KUKA KRL program: MyProgram_033().src

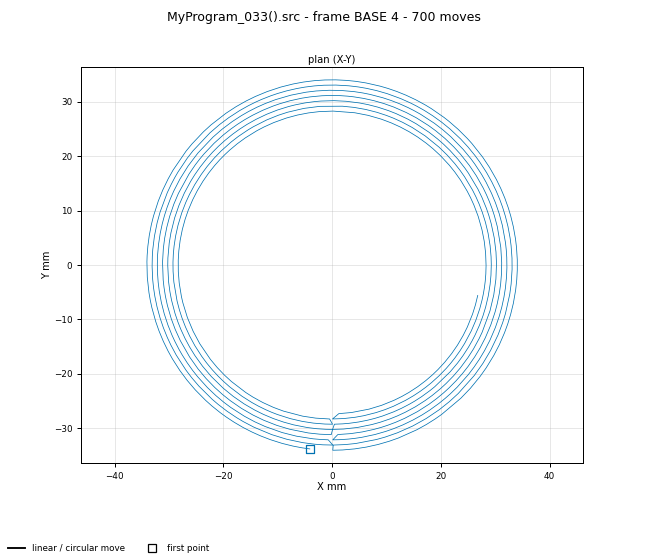
[picture p0: tool path of MyProgram_033().src in frame BASE 4, 700 of 700 moves have a stored position in this frame; points joined in program order, loops and branches not executed]
&ACCESS RVP
&REL 1
&PARAM TEMPLATE = C:\KRC\Roboter\Template\vorgabe
&PARAM EDITMASK = *
DEF MyProgram_033()
; ---- Setting reference (Base) ----
$BASE = BASE_DATA[4]

; --------------------------
; ---- Setting tool (TCP) ----
$TOOL = TOOL_DATA[3]
; --------------------------

$VEL.CP = VEL_APROX_PRINT
Startdeposition()
$VEL.CP = VEL_PRINT
LIN {X -4.1011,Y -33.8077,Z 60,A -103.7519,B 24.8568,C -2.7608,E1 24.9802,E2 -893.1526} C_DIS
LIN {X -5.5425,Y -33.6018,Z 60,A -106.5325,B 24.8572,C -2.7577,E1 24.9725,E2 -890.3623} C_DIS
LIN {X -7.2068,Y -33.2842,Z 60,A -109.5413,B 24.8572,C -2.7571,E1 24.9643,E2 -887.3486} C_DIS
LIN {X -9.1844,Y -32.7935,Z 60,A -113.0761,B 24.8572,C -2.7579,E1 24.9547,E2 -883.8105} C_DIS
LIN {X -11.3943,Y -32.093,Z 60,A -117.2451,B 24.8572,C -2.7582,E1 24.9437,E2 -879.6342} C_DIS
LIN {X -13.2172,Y -31.3861,Z 60,A -119.8941,B 24.8561,C -2.7679,E1 24.9369,E2 -877.0026} C_DIS
LIN {X -14.7733,Y -30.6845,Z 60,A -123.1754,B 24.8561,C -2.767,E1 24.9285,E2 -873.7109} C_DIS
LIN {X -16.3966,Y -29.8493,Z 60,A -126.0085,B 24.8555,C -2.7732,E1 24.9216,E2 -870.8848} C_DIS
LIN {X -18.0247,Y -28.8947,Z 60,A -129.5512,B 24.8555,C -2.7742,E1 24.9131,E2 -867.3333} C_DIS
LIN {X -19.4848,Y -27.931,Z 60,A -132.0562,B 24.8545,C -2.783,E1 24.9073,E2 -864.8412} C_DIS
LIN {X -20.5573,Y -27.1516,Z 60,A -134.7533,B 24.8545,C -2.7823,E1 24.9013,E2 -862.1327} C_DIS
LIN {X -22.102,Y -25.9094,Z 60,A -137.784,B 24.8536,C -2.7913,E1 24.8948,E2 -859.1119} C_DIS
LIN {X -23.2509,Y -24.8836,Z 60,A -140.7805,B 24.8536,C -2.7926,E1 24.8886,E2 -856.1064} C_DIS
LIN {X -25.1661,Y -22.9451,Z 60,A -144.9973,B 24.8521,C -2.8056,E1 24.8805,E2 -851.9024} C_DIS
LIN {X -26.6648,Y -21.1845,Z 60,A -149.0986,B 24.8514,C -2.8125,E1 24.8732,E2 -847.7987} C_DIS
LIN {X -28.0034,Y -19.3806,Z 60,A -153.0848,B 24.8506,C -2.8198,E1 24.8667,E2 -843.8106} C_DIS
LIN {X -29.3744,Y -17.2323,Z 60,A -156.9438,B 24.8491,C -2.8344,E1 24.861,E2 -839.9668} C_DIS
LIN {X -30.1456,Y -15.8438,Z 60,A -159.4556,B 24.8482,C -2.8429,E1 24.8577,E2 -837.4619} C_DIS
LIN {X -31.038,Y -14.0154,Z 60,A -163.101,B 24.8474,C -2.8503,E1 24.8533,E2 -833.8145} C_DIS
LIN {X -31.8171,Y -12.1432,Z 60,A -166.7902,B 24.8466,C -2.8576,E1 24.8495,E2 -830.1221} C_DIS
LIN {X -32.4094,Y -10.4598,Z 60,A -170.2484,B 24.846,C -2.8626,E1 24.8465,E2 -826.656} C_DIS
LIN {X -33.145,Y -7.823,Z 60,A -174.1454,B 24.8439,C -2.882,E1 24.8437,E2 -822.7829} C_DIS
LIN {X -33.441,Y -6.4408,Z 60,A -176.5305,B 24.8432,C -2.8891,E1 24.8424,E2 -820.4008} C_DIS
LIN {X -33.6768,Y -5.0685,Z 60,A -179.4437,B 24.8429,C -2.8917,E1 24.8411,E2 -817.4763} C_DIS
LIN {X -33.9818,Y -2.2443,Z 60,A 175.55,B 24.8415,C -2.9046,E1 24.8399,E2 -812.4709} C_DIS
LIN {X -34.0507,Y 0.5917,Z 60,A 171.6162,B 24.8391,C -2.9263,E1 24.8399,E2 -808.5652} C_DIS
LIN {X -34.0099,Y 1.7604,Z 60,A 169.3433,B 24.8387,C -2.93,E1 24.8401,E2 -806.2875} C_DIS
LIN {X -33.8822,Y 3.4352,Z 60,A 166.5069,B 24.8377,C -2.9387,E1 24.8408,E2 -803.455} C_DIS
LIN {X -33.6225,Y 5.4145,Z 60,A 163.0669,B 24.8366,C -2.9485,E1 24.8422,E2 -800.018} C_DIS
LIN {X -33.2455,Y 7.3857,Z 60,A 159.4228,B 24.8357,C -2.9568,E1 24.8443,E2 -796.3723} C_DIS
LIN {X -32.8452,Y 8.998,Z 60,A 156.7201,B 24.8347,C -2.9662,E1 24.8462,E2 -793.6762} C_DIS
LIN {X -31.9703,Y 11.7339,Z 60,A 151.2142,B 24.8336,C -2.9753,E1 24.8512,E2 -788.161} C_DIS
LIN {X -31.1372,Y 13.7944,Z 60,A 147.9434,B 24.832,C -2.9901,E1 24.8548,E2 -784.9074} C_DIS
LIN {X -30.1384,Y 15.8574,Z 60,A 144.453,B 24.8304,C -3.0042,E1 24.8591,E2 -781.4321} C_DIS
LIN {X -29.2375,Y 17.4636,Z 60,A 140.1056,B 24.8305,C -3.0026,E1 24.8654,E2 -777.0583} C_DIS
LIN {X -26.8529,Y 20.9464,Z 60,A 134.1639,B 24.8273,C -3.0311,E1 24.875,E2 -771.1559} C_DIS
LIN {X -25.7967,Y 22.2333,Z 60,A 130.7426,B 24.8271,C -3.0329,E1 24.8812,E2 -767.7231} C_DIS
LIN {X -23.6637,Y 24.4914,Z 60,A 125.988,B 24.8252,C -3.0493,E1 24.8904,E2 -762.9876} C_DIS
LIN {X -22.2685,Y 25.7663,Z 60,A 122.1842,B 24.825,C -3.0508,E1 24.8984,E2 -759.1724} C_DIS
LIN {X -19.5115,Y 27.912,Z 60,A 116.7582,B 24.8232,C -3.0668,E1 24.9105,E2 -753.7652} C_DIS
LIN {X -17.6615,Y 29.1182,Z 60,A 113.1214,B 24.8223,C -3.0743,E1 24.9191,E2 -750.1348} C_DIS
LIN {X -15.826,Y 30.1549,Z 60,A 109.4298,B 24.8218,C -3.0789,E1 24.9281,E2 -746.4435} C_DIS
LIN {X -14.122,Y 30.9898,Z 60,A 106.4786,B 24.821,C -3.086,E1 24.9356,E2 -743.5019} C_DIS
LIN {X -11.9367,Y 31.8948,Z 60,A 102.2584,B 24.8206,C -3.089,E1 24.9465,E2 -739.2795} C_DIS
LIN {X -9.4384,Y 32.7218,Z 60,A 97.5577,B 24.8204,C -3.0912,E1 24.9591,E2 -734.5758} C_DIS
LIN {X -7.1696,Y 33.2922,Z 60,A 94.1206,B 24.8193,C -3.0998,E1 24.9684,E2 -731.1548} C_DIS
LIN {X -5.2376,Y 33.6506,Z 60,A 90.6316,B 24.8193,C -3.1003,E1 24.978,E2 -727.6635} C_DIS
LIN {X -3.27,Y 33.8982,Z 60,A 87.248,B 24.8191,C -3.1015,E1 24.9874,E2 -724.2808} C_DIS
LIN {X -1.3206,Y 34.0299,Z 60,A 83.9345,B 24.8191,C -3.1024,E1 24.9966,E2 -720.9685} C_DIS
LIN {X 0.6663,Y 34.0493,Z 60,A 80.7843,B 24.8187,C -3.1051,E1 25.0054,E2 -717.825} C_DIS
LIN {X 2.7045,Y 33.9479,Z 60,A 77.3953,B 24.8187,C -3.1056,E1 25.0148,E2 -714.4386} C_DIS
LIN {X 4.3939,Y 33.771,Z 60,A 74.5416,B 24.8187,C -3.1052,E1 25.0227,E2 -711.5859} C_DIS
LIN {X 6.2336,Y 33.4806,Z 60,A 70.9287,B 24.8195,C -3.0986,E1 25.0327,E2 -707.9612} C_DIS
LIN {X 8.817,Y 32.8943,Z 60,A 66.9146,B 24.8192,C -3.1013,E1 25.0435,E2 -703.9594} C_DIS
LIN {X 10.2829,Y 32.4658,Z 60,A 64.544,B 24.8192,C -3.1018,E1 25.0499,E2 -701.5942} C_DIS
LIN {X 11.8741,Y 31.9182,Z 60,A 61.4166,B 24.8198,C -3.0958,E1 25.0581,E2 -698.4589} C_DIS
LIN {X 13.5855,Y 31.2283,Z 60,A 58.3959,B 24.8201,C -3.0937,E1 25.0659,E2 -695.4401} C_DIS
LIN {X 15.3952,Y 30.3775,Z 60,A 54.9755,B 24.8206,C -3.0889,E1 25.0745,E2 -692.0176} C_DIS
LIN {X 17.1475,Y 29.4242,Z 60,A 51.9399,B 24.8206,C -3.0884,E1 25.0819,E2 -688.9897} C_DIS
LIN {X 18.2192,Y 28.7727,Z 60,A 49.141,B 24.8221,C -3.0765,E1 25.0885,E2 -686.1715} C_DIS
LIN {X 20.5404,Y 27.1644,Z 60,A 45.1493,B 24.8218,C -3.0784,E1 25.0975,E2 -682.1983} C_DIS
LIN {X 21.455,Y 26.4477,Z 60,A 42.9139,B 24.8227,C -3.0713,E1 25.1024,E2 -679.9543} C_DIS
LIN {X 23.1922,Y 24.9385,Z 60,A 38.6625,B 24.8241,C -3.0588,E1 25.1113,E2 -675.6903} C_DIS
LIN {X 24.8778,Y 23.2567,Z 60,A 35.3372,B 24.8241,C -3.0594,E1 25.1177,E2 -672.3807} C_DIS
LIN {X 25.686,Y 22.3614,Z 60,A 32.55,B 24.8257,C -3.0448,E1 25.1229,E2 -669.5713} C_DIS
LIN {X 27.6713,Y 19.852,Z 60,A 28.2174,B 24.8255,C -3.0464,E1 25.1303,E2 -665.2631} C_DIS
LIN {X 28.9223,Y 17.9798,Z 60,A 23.4081,B 24.8282,C -3.0228,E1 25.1376,E2 -660.422} C_DIS
LIN {X 30.1935,Y 15.7523,Z 60,A 19.4635,B 24.829,C -3.0166,E1 25.1429,E2 -656.4831} C_DIS
LIN {X 31.019,Y 14.0575,Z 60,A 16.5637,B 24.8295,C -3.0117,E1 25.1463,E2 -653.5874} C_DIS
LIN {X 31.744,Y 12.3327,Z 60,A 13.1959,B 24.8309,C -2.9997,E1 25.1499,E2 -650.2098} C_DIS
LIN {X 32.3816,Y 10.5466,Z 60,A 10.2406,B 24.8315,C -2.9938,E1 25.1525,E2 -647.2573} C_DIS
LIN {X 32.847,Y 8.9926,Z 60,A 7.5063,B 24.8325,C -2.9857,E1 25.1546,E2 -644.5194} C_DIS
LIN {X 33.3186,Y 7.0474,Z 60,A 3.8113,B 24.8341,C -2.9709,E1 25.1569,E2 -640.8108} C_DIS
LIN {X 33.7159,Y 4.7991,Z 60,A 0.1976,B 24.8351,C -2.9624,E1 25.1585,E2 -637.1983} C_DIS
LIN {X 33.9025,Y 3.2253,Z 60,A -2.4984,B 24.836,C -2.9537,E1 25.1593,E2 -634.4977} C_DIS
LIN {X 34.0412,Y 0.9926,Z 60,A -6.0206,B 24.837,C -2.9455,E1 25.1598,E2 -630.977} C_DIS
LIN {X 34.043,Y -0.9308,Z 60,A -9.3922,B 24.8383,C -2.9334,E1 25.1596,E2 -627.5968} C_DIS
LIN {X 33.9493,Y -2.6804,Z 60,A -12.2431,B 24.8392,C -2.9256,E1 25.1591,E2 -624.7443} C_DIS
LIN {X 33.7459,Y -4.5841,Z 60,A -15.5123,B 24.8404,C -2.9148,E1 25.158,E2 -621.4688} C_DIS
LIN {X 33.3196,Y -7.0427,Z 60,A -19.7936,B 24.8419,C -2.9005,E1 25.1558,E2 -617.1788} C_DIS
LIN {X 32.8125,Y -9.1163,Z 60,A -23.0848,B 24.8427,C -2.8938,E1 25.1535,E2 -613.8906} C_DIS
LIN {X 32.296,Y -10.8043,Z 60,A -25.7379,B 24.8431,C -2.8893,E1 25.1512,E2 -611.2421} C_DIS
LIN {X 31.7073,Y -12.4251,Z 60,A -28.7099,B 24.8442,C -2.8796,E1 25.1483,E2 -608.2636} C_DIS
LIN {X 30.7314,Y -14.6755,Z 60,A -33.9408,B 24.8472,C -2.8517,E1 25.1422,E2 -602.9951} C_DIS
LIN {X 29.7216,Y -16.626,Z 60,A -37.262,B 24.8478,C -2.8465,E1 25.1378,E2 -599.6788} C_DIS
LIN {X 28.3176,Y -18.9173,Z 60,A -41.1609,B 24.8482,C -2.8428,E1 25.1319,E2 -595.7907} C_DIS
LIN {X 27.2015,Y -20.4909,Z 60,A -44.1382,B 24.8487,C -2.8379,E1 25.1271,E2 -592.8163} C_DIS
LIN {X 25.4199,Y -22.6633,Z 60,A -49.9904,B 24.8516,C -2.8103,E1 25.1164,E2 -586.9256} C_DIS
LIN {X 23.6533,Y -24.5014,Z 60,A -54.523,B 24.853,C -2.797,E1 25.1074,E2 -582.3803} C_DIS
LIN {X 20.127,Y -27.4718,Z 60,A -60.5922,B 24.8524,C -2.8031,E1 25.0943,E2 -576.3485} C_DIS
LIN {X 18.9319,Y -28.3082,Z 60,A -63.281,B 24.8532,C -2.7951,E1 25.0881,E2 -573.65} C_DIS
LIN {X 17.3293,Y -29.3171,Z 60,A -67.2414,B 24.8549,C -2.7791,E1 25.0786,E2 -569.664} C_DIS
LIN {X 15.5543,Y -30.2963,Z 60,A -70.9708,B 24.8559,C -2.7694,E1 25.0693,E2 -565.922} C_DIS
LIN {X 12.179,Y -31.8037,Z 60,A -76.2659,B 24.8556,C -2.7723,E1 25.0558,E2 -560.6462} C_DIS
LIN {X 10.5249,Y -32.3887,Z 60,A -79.589,B 24.8565,C -2.764,E1 25.0469,E2 -557.31} C_DIS
LIN {X 8.4575,Y -32.9886,Z 60,A -83.2845,B 24.857,C -2.7593,E1 25.037,E2 -553.6093} C_DIS
LIN {X 6.2909,Y -33.4695,Z 60,A -86.7215,B 24.857,C -2.7598,E1 25.0276,E2 -550.1776} C_DIS
LIN {X 4.1516,Y -33.8017,Z 60,A -90.2648,B 24.857,C -2.7585,E1 25.0178,E2 -546.6345} C_DIS
LIN {X 1.9064,Y -34.0016,Z 60,A -94.0756,B 24.8573,C -2.7566,E1 25.0072,E2 -542.8209} C_DIS
LIN {X 0.1202,Y -34.0515,Z 60,A -95.9136,B 24.8559,C -2.7694,E1 25.0021,E2 -541.0138} C_DIS
Enddeposition()
LIN {X 0.1202,Y -34.0515,Z 60,A -95.9136,B 24.8559,C -2.7694,E1 25.0021,E2 -541.0138} C_DIS
Startdeposition()
$VEL.CP = VEL_PRINT
LIN {X 0.2045,Y -33.097,Z 60,A -95.4369,B 24.8538,C -2.7896,E1 25.0036,E2 -541.5385} C_DIS
LIN {X 2.3595,Y -33.0129,Z 60,A -91.3479,B 24.8532,C -2.7953,E1 25.015,E2 -545.6395} C_DIS
LIN {X 4.3325,Y -32.8127,Z 60,A -87.4957,B 24.8525,C -2.8025,E1 25.0257,E2 -549.5057} C_DIS
LIN {X 8.1456,Y -32.0792,Z 60,A -81.9514,B 24.8534,C -2.7939,E1 25.0408,E2 -555.0225} C_DIS
LIN {X 9.7251,Y -31.6363,Z 60,A -78.376,B 24.8521,C -2.8062,E1 25.0504,E2 -558.6209} C_DIS
LIN {X 12.006,Y -30.843,Z 60,A -74.0706,B 24.8513,C -2.8132,E1 25.0617,E2 -562.9339} C_DIS
LIN {X 14.8198,Y -29.5942,Z 60,A -69.0859,B 24.8509,C -2.8169,E1 25.0743,E2 -567.9146} C_DIS
LIN {X 17.289,Y -28.2232,Z 60,A -63.6869,B 24.8493,C -2.8323,E1 25.0874,E2 -573.3336} C_DIS
LIN {X 19.6801,Y -26.6116,Z 60,A -59.6968,B 24.8497,C -2.8288,E1 25.0964,E2 -577.3018} C_DIS
LIN {X 21.5621,Y -25.1105,Z 60,A -54.3541,B 24.847,C -2.8538,E1 25.108,E2 -582.6832} C_DIS
LIN {X 23.1978,Y -23.6076,Z 60,A -50.3874,B 24.8458,C -2.8645,E1 25.1159,E2 -586.6586} C_DIS
LIN {X 26.126,Y -20.3201,Z 60,A -43.8899,B 24.8455,C -2.868,E1 25.1276,E2 -593.1349} C_DIS
LIN {X 27.705,Y -18.1078,Z 60,A -38.537,B 24.8431,C -2.8899,E1 25.1361,E2 -598.5131} C_DIS
LIN {X 29.1251,Y -15.7222,Z 60,A -33.8097,B 24.8417,C -2.9024,E1 25.1426,E2 -603.2454} C_DIS
LIN {X 30.4955,Y -12.8635,Z 60,A -28.9128,B 24.8409,C -2.91,E1 25.1482,E2 -608.1339} C_DIS
LIN {X 31.3542,Y -10.6002,Z 60,A -24.761,B 24.8395,C -2.9221,E1 25.1522,E2 -612.2911} C_DIS
LIN {X 31.8641,Y -8.9501,Z 60,A -21.1192,B 24.8375,C -2.9407,E1 25.155,E2 -615.9559} C_DIS
LIN {X 32.6625,Y -5.3501,Z 60,A -15.7724,B 24.837,C -2.9455,E1 25.1579,E2 -621.283} C_DIS
LIN {X 32.9129,Y -3.4907,Z 60,A -11.951,B 24.8349,C -2.964,E1 25.1592,E2 -625.1255} C_DIS
LIN {X 33.0886,Y -0.7895,Z 60,A -7.3415,B 24.8334,C -2.9775,E1 25.1598,E2 -629.7397} C_DIS
LIN {X 33.0726,Y 1.2789,Z 60,A -3.8158,B 24.8322,C -2.9879,E1 25.1595,E2 -633.269} C_DIS
LIN {X 32.9048,Y 3.567,Z 60,A -0.295,B 24.8316,C -2.9937,E1 25.1586,E2 -636.7827} C_DIS
LIN {X 32.7236,Y 4.9627,Z 60,A 2.3683,B 24.8303,C -3.0044,E1 25.1576,E2 -639.4557} C_DIS
LIN {X 32.3321,Y 7.0767,Z 60,A 5.9021,B 24.8294,C -3.013,E1 25.1557,E2 -642.9891} C_DIS
LIN {X 31.8536,Y 8.9878,Z 60,A 9.2415,B 24.8283,C -3.0221,E1 25.1533,E2 -646.3309} C_DIS
LIN {X 31.334,Y 10.6598,Z 60,A 12.4134,B 24.8271,C -3.0329,E1 25.1505,E2 -649.5104} C_DIS
LIN {X 30.8145,Y 12.0789,Z 60,A 14.7067,B 24.8268,C -3.0358,E1 25.1483,E2 -651.7979} C_DIS
LIN {X 30.1671,Y 13.6158,Z 60,A 17.9721,B 24.8252,C -3.0492,E1 25.1446,E2 -655.077} C_DIS
LIN {X 29.3671,Y 15.2653,Z 60,A 20.8782,B 24.8247,C -3.054,E1 25.141,E2 -657.9791} C_DIS
LIN {X 28.3881,Y 17.0175,Z 60,A 24.7982,B 24.8229,C -3.0692,E1 25.1355,E2 -661.9149} C_DIS
LIN {X 27.1221,Y 18.9699,Z 60,A 27.9977,B 24.8231,C -3.0679,E1 25.1305,E2 -665.0953} C_DIS
LIN {X 26.2731,Y 20.1291,Z 60,A 31.0095,B 24.8216,C -3.0809,E1 25.1255,E2 -668.1236} C_DIS
LIN {X 24.9894,Y 21.7024,Z 60,A 34.3231,B 24.8209,C -3.0861,E1 25.1195,E2 -671.4345} C_DIS
LIN {X 23.6198,Y 23.1855,Z 60,A 38.4346,B 24.8191,C -3.1018,E1 25.1115,E2 -675.5653} C_DIS
LIN {X 21.6787,Y 25.0098,Z 60,A 42.4056,B 24.8191,C -3.1023,E1 25.1034,E2 -679.5217} C_DIS
LIN {X 20.1341,Y 26.2693,Z 60,A 46.2217,B 24.8178,C -3.1132,E1 25.095,E2 -683.3494} C_DIS
LIN {X 18.4879,Y 27.4526,Z 60,A 49.4342,B 24.8176,C -3.1151,E1 25.0876,E2 -686.5553} C_DIS
LIN {X 16.9247,Y 28.4433,Z 60,A 52.4596,B 24.8173,C -3.1176,E1 25.0804,E2 -689.577} C_DIS
LIN {X 15.6004,Y 29.1906,Z 60,A 54.8557,B 24.8172,C -3.1181,E1 25.0746,E2 -691.9675} C_DIS
LIN {X 14.4137,Y 29.7944,Z 60,A 57.4788,B 24.8164,C -3.1249,E1 25.068,E2 -694.5996} C_DIS
LIN {X 12.61,Y 30.6015,Z 60,A 61.2733,B 24.8154,C -3.133,E1 25.0582,E2 -698.4043} C_DIS
LIN {X 10.1317,Y 31.5084,Z 60,A 65.3664,B 24.8157,C -3.1312,E1 25.0475,E2 -702.4849} C_DIS
LIN {X 8.2097,Y 32.063,Z 60,A 69.151,B 24.8149,C -3.1371,E1 25.0373,E2 -706.2776} C_DIS
LIN {X 6.3041,Y 32.4916,Z 60,A 72.3612,B 24.815,C -3.1367,E1 25.0285,E2 -709.4826} C_DIS
LIN {X 4.8128,Y 32.7461,Z 60,A 74.7387,B 24.8152,C -3.1347,E1 25.022,E2 -711.8532} C_DIS
LIN {X 3.0706,Y 32.9547,Z 60,A 78.3371,B 24.8144,C -3.1414,E1 25.0119,E2 -715.4651} C_DIS
LIN {X 0.6892,Y 33.0906,Z 60,A 82.3493,B 24.8146,C -3.1398,E1 25.0008,E2 -719.4724} C_DIS
LIN {X -1.5064,Y 33.0631,Z 60,A 85.9149,B 24.8151,C -3.1362,E1 24.9908,E2 -723.0299} C_DIS
LIN {X -3.2719,Y 32.9353,Z 60,A 89.2096,B 24.8149,C -3.1372,E1 24.9817,E2 -726.3286} C_DIS
LIN {X -5.02,Y 32.7148,Z 60,A 91.7867,B 24.8157,C -3.1304,E1 24.9746,E2 -728.8915} C_DIS
LIN {X -6.5185,Y 32.4493,Z 60,A 94.6895,B 24.8157,C -3.1311,E1 24.9666,E2 -731.7991} C_DIS
LIN {X -8.3984,Y 32.0142,Z 60,A 98.2278,B 24.8157,C -3.13,E1 24.957,E2 -735.3397} C_DIS
LIN {X -10.0341,Y 31.5395,Z 60,A 100.7953,B 24.8166,C -3.123,E1 24.9502,E2 -737.8948} C_DIS
LIN {X -11.274,Y 31.118,Z 60,A 103.5496,B 24.8164,C -3.125,E1 24.9429,E2 -740.6594} C_DIS
LIN {X -12.9995,Y 30.4377,Z 60,A 106.309,B 24.8174,C -3.1162,E1 24.9358,E2 -743.404} C_DIS
LIN {X -14.1215,Y 29.9343,Z 60,A 108.4303,B 24.8178,C -3.113,E1 24.9304,E2 -745.5229} C_DIS
LIN {X -15.3884,Y 29.3025,Z 60,A 110.9912,B 24.8181,C -3.1101,E1 24.9241,E2 -748.0839} C_DIS
LIN {X -17.0304,Y 28.3798,Z 60,A 114.8593,B 24.8181,C -3.1101,E1 24.9147,E2 -751.9636} C_DIS
LIN {X -19.006,Y 27.0964,Z 60,A 118.1285,B 24.8199,C -3.095,E1 24.9072,E2 -755.2074} C_DIS
LIN {X -20.7047,Y 25.8224,Z 60,A 122.9494,B 24.8196,C -3.0977,E1 24.8965,E2 -760.0525} C_DIS
LIN {X -22.4758,Y 24.2961,Z 60,A 127.3905,B 24.8202,C -3.0921,E1 24.8874,E2 -764.4982} C_DIS
LIN {X -25.5874,Y 20.9946,Z 60,A 134.3352,B 24.8234,C -3.0648,E1 24.8745,E2 -771.4087} C_DIS
LIN {X -26.6205,Y 19.6678,Z 60,A 137.6287,B 24.8239,C -3.0605,E1 24.869,E2 -774.7075} C_DIS
LIN {X -28.3514,Y 17.0781,Z 60,A 142.2081,B 24.8264,C -3.0389,E1 24.8621,E2 -779.2585} C_DIS
LIN {X -28.9377,Y 16.0644,Z 60,A 144.4768,B 24.8268,C -3.0352,E1 24.859,E2 -781.5302} C_DIS
LIN {X -29.5648,Y 14.8797,Z 60,A 146.7395,B 24.8276,C -3.0281,E1 24.8561,E2 -783.7879} C_DIS
LIN {X -30.3082,Y 13.2994,Z 60,A 150.7686,B 24.8277,C -3.0275,E1 24.8515,E2 -787.8377} C_DIS
LIN {X -31.6393,Y 9.7155,Z 60,A 156.2309,B 24.8311,C -2.9982,E1 24.8465,E2 -793.2608} C_DIS
LIN {X -32.1756,Y 7.7552,Z 60,A 160.4111,B 24.8317,C -2.9927,E1 24.8436,E2 -797.4522} C_DIS
LIN {X -32.6737,Y 5.2775,Z 60,A 165.1809,B 24.8328,C -2.9822,E1 24.8412,E2 -802.2253} C_DIS
LIN {X -32.973,Y 2.8674,Z 60,A 168.4595,B 24.8352,C -2.9617,E1 24.8403,E2 -805.4743} C_DIS
LIN {X -33.057,Y 1.6305,Z 60,A 170.8713,B 24.8357,C -2.9571,E1 24.8399,E2 -807.8897} C_DIS
LIN {X -33.096,Y -0.2924,Z 60,A 174.4282,B 24.8366,C -2.9485,E1 24.8399,E2 -811.4474} C_DIS
LIN {X -32.9885,Y -2.6819,Z 60,A 178.201,B 24.8384,C -2.9327,E1 24.8404,E2 -815.2051} C_DIS
LIN {X -32.8369,Y -4.146,Z 60,A -179.0925,B 24.8391,C -2.9261,E1 24.8413,E2 -817.9121} C_DIS
LIN {X -32.594,Y -5.7529,Z 60,A -176.0974,B 24.8399,C -2.919,E1 24.8427,E2 -820.908} C_DIS
LIN {X -32.1918,Y -7.6888,Z 60,A -172.6651,B 24.841,C -2.9088,E1 24.8447,E2 -824.3361} C_DIS
LIN {X -31.643,Y -9.7037,Z 60,A -169.103,B 24.8422,C -2.8978,E1 24.8475,E2 -827.8923} C_DIS
LIN {X -31.0365,Y -11.4963,Z 60,A -165.5855,B 24.843,C -2.8904,E1 24.8508,E2 -831.412} C_DIS
LIN {X -30.3151,Y -13.2835,Z 60,A -162.7793,B 24.8445,C -2.8766,E1 24.8538,E2 -834.2009} C_DIS
LIN {X -29.6522,Y -14.7033,Z 60,A -159.5325,B 24.8448,C -2.8737,E1 24.8577,E2 -837.4584} C_DIS
LIN {X -28.67,Y -16.5374,Z 60,A -155.4519,B 24.8454,C -2.8684,E1 24.8633,E2 -841.5477} C_DIS
LIN {X -26.8802,Y -19.3109,Z 60,A -150.7238,B 24.8479,C -2.8457,E1 24.8706,E2 -846.2449} C_DIS
LIN {X -25.8421,Y -20.6801,Z 60,A -146.7435,B 24.8477,C -2.8477,E1 24.8775,E2 -850.2488} C_DIS
LIN {X -24.4962,Y -22.2575,Z 60,A -143.0433,B 24.8484,C -2.8408,E1 24.8844,E2 -853.9493} C_DIS
LIN {X -22.0604,Y -24.6738,Z 60,A -138.1883,B 24.8507,C -2.8189,E1 24.8941,E2 -858.7721} C_DIS
LIN {X -20.9813,Y -25.598,Z 60,A -135.1647,B 24.8507,C -2.8197,E1 24.9006,E2 -861.809} C_DIS
LIN {X -19.3358,Y -26.8623,Z 60,A -131.5019,B 24.8512,C -2.8143,E1 24.9088,E2 -865.4721} C_DIS
LIN {X -17.5879,Y -28.0377,Z 60,A -128.1825,B 24.8521,C -2.8056,E1 24.9165,E2 -868.7814} C_DIS
LIN {X -16.3357,Y -28.7859,Z 60,A -125.413,B 24.8523,C -2.8045,E1 24.9232,E2 -871.5566} C_DIS
LIN {X -14.3684,Y -29.8161,Z 60,A -120.9727,B 24.8521,C -2.8059,E1 24.9343,E2 -876.0121} C_DIS
LIN {X -11.0977,Y -31.1814,Z 60,A -114.7027,B 24.8525,C -2.8017,E1 24.9507,E2 -882.2853} C_DIS
LIN {X -8.3337,Y -32.0312,Z 60,A -109.9263,B 24.8531,C -2.7961,E1 24.9635,E2 -887.0559} C_DIS
LIN {X -5.4058,Y -32.6532,Z 60,A -105.0089,B 24.8536,C -2.7913,E1 24.9769,E2 -891.9672} C_DIS
LIN {X -3.2219,Y -32.9404,Z 60,A -101.8852,B 24.8545,C -2.7831,E1 24.9856,E2 -895.0735} C_DIS
LIN {X -1.6841,Y -33.0544,Z 60,A -98.863,B 24.8541,C -2.7871,E1 24.994,E2 -898.1063} C_DIS
LIN {X 0.1302,Y -33.0962,Z 60,A -97.1686,B 24.8557,C -2.7713,E1 24.9987,E2 -899.7633} C_DIS
Enddeposition()
LIN {X 0.1302,Y -33.0962,Z 60,A -97.1686,B 24.8557,C -2.7713,E1 24.9987,E2 -899.7633} C_DIS
Startdeposition()
$VEL.CP = VEL_PRINT
LIN {X -0.7153,Y -32.1318,Z 60,A -98.6258,B 24.854,C -2.7884,E1 24.9947,E2 -898.3466} C_DIS
LIN {X -2.0689,Y -32.0727,Z 60,A -100.8693,B 24.8538,C -2.7901,E1 24.9884,E2 -896.1066} C_DIS
LIN {X -3.5101,Y -31.9474,Z 60,A -103.7174,B 24.854,C -2.7874,E1 24.9805,E2 -893.2506} C_DIS
LIN {X -6.5606,Y -31.463,Z 60,A -110.1953,B 24.8549,C -2.7794,E1 24.9626,E2 -886.7468} C_DIS
LIN {X -9.1763,Y -30.8007,Z 60,A -114.641,B 24.8542,C -2.7861,E1 24.9507,E2 -882.3099} C_DIS
LIN {X -12.3035,Y -29.6913,Z 60,A -119.3861,B 24.8524,C -2.8026,E1 24.9384,E2 -877.5946} C_DIS
LIN {X -14.2126,Y -28.8258,Z 60,A -123.9875,B 24.8529,C -2.7986,E1 24.9267,E2 -872.972} C_DIS
LIN {X -16.1045,Y -27.8137,Z 60,A -128.1219,B 24.8526,C -2.8009,E1 24.9166,E2 -868.8309} C_DIS
LIN {X -18.6436,Y -26.1794,Z 60,A -132.797,B 24.8511,C -2.8156,E1 24.9058,E2 -864.1755} C_DIS
LIN {X -19.882,Y -25.2519,Z 60,A -135.745,B 24.8507,C -2.8187,E1 24.8993,E2 -861.2242} C_DIS
LIN {X -21.3807,Y -23.9963,Z 60,A -139.2884,B 24.8501,C -2.8247,E1 24.8918,E2 -857.6813} C_DIS
LIN {X -22.9252,Y -22.5252,Z 60,A -143.5033,B 24.8497,C -2.829,E1 24.8834,E2 -853.4589} C_DIS
LIN {X -24.7375,Y -20.5185,Z 60,A -147.746,B 24.848,C -2.8444,E1 24.8757,E2 -849.234} C_DIS
LIN {X -25.6401,Y -19.379,Z 60,A -150.286,B 24.8473,C -2.8509,E1 24.8713,E2 -846.6974} C_DIS
LIN {X -26.6364,Y -17.9848,Z 60,A -153.6792,B 24.8468,C -2.8556,E1 24.8659,E2 -843.2987} C_DIS
LIN {X -27.5573,Y -16.5395,Z 60,A -156.5093,B 24.8458,C -2.8652,E1 24.8618,E2 -840.477} C_DIS
LIN {X -28.1696,Y -15.4743,Z 60,A -158.7932,B 24.8452,C -2.8702,E1 24.8587,E2 -838.1931} C_DIS
LIN {X -28.8992,Y -14.0622,Z 60,A -161.3805,B 24.8442,C -2.8797,E1 24.8554,E2 -835.6148} C_DIS
LIN {X -29.4323,Y -12.9111,Z 60,A -164.1998,B 24.844,C -2.8816,E1 24.8522,E2 -832.7845} C_DIS
LIN {X -30.1822,Y -11.0442,Z 60,A -167.4588,B 24.8426,C -2.8943,E1 24.8489,E2 -829.5376} C_DIS
LIN {X -30.8706,Y -8.9417,Z 60,A -172.0182,B 24.8418,C -2.9012,E1 24.8452,E2 -824.9684} C_DIS
LIN {X -31.4046,Y -6.8329,Z 60,A -175.525,B 24.8403,C -2.9156,E1 24.843,E2 -821.4755} C_DIS
LIN {X -31.7843,Y -4.7678,Z 60,A -178.7753,B 24.8386,C -2.9306,E1 24.8414,E2 -818.2419} C_DIS
LIN {X -31.9804,Y -3.1964,Z 60,A 178.3793,B 24.8377,C -2.9391,E1 24.8405,E2 -815.3999} C_DIS
LIN {X -32.1078,Y -1.4183,Z 60,A 174.6768,B 24.837,C -2.9451,E1 24.8398,E2 -811.6893} C_DIS
LIN {X -32.1379,Y 0.2156,Z 60,A 172.0129,B 24.8358,C -2.956,E1 24.8398,E2 -809.0356} C_DIS
LIN {X -32.0787,Y 1.9696,Z 60,A 168.7941,B 24.8348,C -2.9651,E1 24.8402,E2 -805.8193} C_DIS
LIN {X -31.9124,Y 3.8118,Z 60,A 165.224,B 24.8338,C -2.9734,E1 24.8412,E2 -802.2476} C_DIS
LIN {X -31.6091,Y 5.8156,Z 60,A 161.6312,B 24.8326,C -2.9848,E1 24.8429,E2 -798.6608} C_DIS
LIN {X -31.2255,Y 7.6094,Z 60,A 158.365,B 24.8314,C -2.9949,E1 24.8449,E2 -795.3996} C_DIS
LIN {X -30.8172,Y 9.1232,Z 60,A 155.8063,B 24.8302,C -3.0052,E1 24.8468,E2 -792.8507} C_DIS
LIN {X -30.3452,Y 10.5875,Z 60,A 152.8019,B 24.8295,C -3.0116,E1 24.8495,E2 -789.8443} C_DIS
LIN {X -29.7422,Y 12.1789,Z 60,A 149.6558,B 24.8286,C -3.0198,E1 24.8527,E2 -786.7002} C_DIS
LIN {X -29.1245,Y 13.5905,Z 60,A 146.9426,B 24.8277,C -3.028,E1 24.8559,E2 -783.992} C_DIS
LIN {X -27.9696,Y 15.8309,Z 60,A 142.1992,B 24.8264,C -3.0389,E1 24.8621,E2 -779.2496} C_DIS
LIN {X -26.466,Y 18.2338,Z 60,A 136.5813,B 24.8253,C -3.0483,E1 24.8708,E2 -773.626} C_DIS
LIN {X -24.6789,Y 20.5889,Z 60,A 131.1092,B 24.824,C -3.0602,E1 24.8804,E2 -768.1569} C_DIS
LIN {X -21.891,Y 23.5318,Z 60,A 124.8467,B 24.8211,C -3.085,E1 24.8926,E2 -761.9269} C_DIS
LIN {X -20.2021,Y 24.9965,Z 60,A 120.4479,B 24.8205,C -3.0902,E1 24.902,E2 -757.5236} C_DIS
LIN {X -18.3745,Y 26.3691,Z 60,A 116.6627,B 24.8192,C -3.1007,E1 24.9106,E2 -753.7504} C_DIS
LIN {X -16.6745,Y 27.4755,Z 60,A 113.2127,B 24.8183,C -3.1088,E1 24.9187,E2 -750.3086} C_DIS
LIN {X -15.3521,Y 28.2359,Z 60,A 110.265,B 24.818,C -3.1113,E1 24.9259,E2 -747.3585} C_DIS
LIN {X -13.8092,Y 29.0216,Z 60,A 107.2908,B 24.8173,C -3.1171,E1 24.9333,E2 -744.3903} C_DIS
LIN {X -12.2881,Y 29.6966,Z 60,A 103.8696,B 24.8173,C -3.1171,E1 24.9421,E2 -740.9614} C_DIS
LIN {X -10.3903,Y 30.4138,Z 60,A 100.0066,B 24.8171,C -3.1193,E1 24.9523,E2 -737.0959} C_DIS
LIN {X -7.5813,Y 31.2322,Z 60,A 95.0969,B 24.8161,C -3.1274,E1 24.9655,E2 -732.1981} C_DIS
LIN {X -4.8177,Y 31.7765,Z 60,A 90.8046,B 24.8148,C -3.1382,E1 24.9772,E2 -727.9272} C_DIS
LIN {X -2.9177,Y 32.0061,Z 60,A 86.7045,B 24.8154,C -3.1332,E1 24.9887,E2 -723.8125} C_DIS
LIN {X -0.5298,Y 32.1352,Z 60,A 82.2698,B 24.8154,C -3.1327,E1 25.001,E2 -719.3761} C_DIS
LIN {X 1.6757,Y 32.0955,Z 60,A 78.4348,B 24.8154,C -3.134,E1 25.0117,E2 -715.5452} C_DIS
LIN {X 4.085,Y 31.8788,Z 60,A 74.6069,B 24.8148,C -3.1386,E1 25.0223,E2 -711.7307} C_DIS
LIN {X 5.6076,Y 31.6467,Z 60,A 71.8608,B 24.8148,C -3.1377,E1 25.0299,E2 -708.9853} C_DIS
LIN {X 6.9631,Y 31.3764,Z 60,A 68.9821,B 24.8156,C -3.132,E1 25.0378,E2 -706.0968} C_DIS
LIN {X 9.3593,Y 30.7464,Z 60,A 65.1991,B 24.8151,C -3.1363,E1 25.0479,E2 -702.33} C_DIS
LIN {X 10.8355,Y 30.2577,Z 60,A 62.148,B 24.8157,C -3.1308,E1 25.056,E2 -699.2719} C_DIS
LIN {X 12.413,Y 29.6454,Z 60,A 59.3663,B 24.8157,C -3.1306,E1 25.0632,E2 -696.4959} C_DIS
LIN {X 13.9702,Y 28.9444,Z 60,A 56.3307,B 24.8161,C -3.1272,E1 25.0709,E2 -693.46} C_DIS
LIN {X 15.0022,Y 28.4231,Z 60,A 54.1232,B 24.8166,C -3.1229,E1 25.0764,E2 -691.2484} C_DIS
LIN {X 16.2191,Y 27.7471,Z 60,A 51.0142,B 24.8179,C -3.112,E1 25.0839,E2 -688.1228} C_DIS
LIN {X 18.7648,Y 26.0924,Z 60,A 46.4958,B 24.8176,C -3.1143,E1 25.0944,E2 -683.6251} C_DIS
LIN {X 20.337,Y 24.8871,Z 60,A 42.3714,B 24.8192,C -3.1007,E1 25.1034,E2 -679.4837} C_DIS
LIN {X 21.8429,Y 23.5767,Z 60,A 38.334,B 24.8207,C -3.0878,E1 25.1118,E2 -675.432} C_DIS
LIN {X 24.0952,Y 21.2691,Z 60,A 33.1077,B 24.8214,C -3.0821,E1 25.1218,E2 -670.215} C_DIS
LIN {X 25.4626,Y 19.6114,Z 60,A 29.3914,B 24.8223,C -3.0747,E1 25.1282,E2 -666.4985} C_DIS
LIN {X 26.2596,Y 18.5308,Z 60,A 26.7666,B 24.8233,C -3.0659,E1 25.1325,E2 -663.8656} C_DIS
LIN {X 27.4745,Y 16.6753,Z 60,A 23.3272,B 24.8237,C -3.0626,E1 25.1376,E2 -660.4358} C_DIS
LIN {X 28.2947,Y 15.2435,Z 60,A 20.1887,B 24.8249,C -3.0523,E1 25.1419,E2 -657.2891} C_DIS
LIN {X 29.3,Y 13.2079,Z 60,A 15.7928,B 24.8267,C -3.0366,E1 25.1471,E2 -652.8797} C_DIS
LIN {X 30.0387,Y 11.4288,Z 60,A 12.6901,B 24.8273,C -3.0313,E1 25.1503,E2 -649.7817} C_DIS
LIN {X 30.7079,Y 9.4845,Z 60,A 8.9747,B 24.8286,C -3.0199,E1 25.1535,E2 -646.0605} C_DIS
LIN {X 31.3054,Y 7.2744,Z 60,A 4.5208,B 24.8305,C -3.0027,E1 25.1565,E2 -641.5916} C_DIS
LIN {X 31.8734,Y 4.1239,Z 60,A -0.0277,B 24.8307,C -3.0012,E1 25.1586,E2 -637.0661} C_DIS
LIN {X 32.0205,Y 2.7619,Z 60,A -2.7122,B 24.8319,C -2.9903,E1 25.1593,E2 -634.3717} C_DIS
LIN {X 32.1089,Y 1.3993,Z 60,A -5.2676,B 24.833,C -2.981,E1 25.1597,E2 -631.8096} C_DIS
LIN {X 32.1356,Y -0.5008,Z 60,A -8.7386,B 24.8343,C -2.9693,E1 25.1597,E2 -628.3314} C_DIS
LIN {X 32.0631,Y -2.2144,Z 60,A -11.8385,B 24.8354,C -2.9591,E1 25.1592,E2 -625.2259} C_DIS
LIN {X 31.8561,Y -4.2576,Z 60,A -15.3207,B 24.8364,C -2.9501,E1 25.1581,E2 -621.7431} C_DIS
LIN {X 31.589,Y -5.9233,Z 60,A -18.2147,B 24.8373,C -2.9423,E1 25.1567,E2 -618.8475} C_DIS
LIN {X 31.1975,Y -7.7244,Z 60,A -21.8323,B 24.8389,C -2.9276,E1 25.1544,E2 -615.216} C_DIS
LIN {X 30.7173,Y -9.4538,Z 60,A -24.5603,B 24.8393,C -2.9243,E1 25.1523,E2 -612.4958} C_DIS
LIN {X 30.0155,Y -11.4878,Z 60,A -28.9749,B 24.8414,C -2.9048,E1 25.1481,E2 -608.0598} C_DIS
LIN {X 29.0156,Y -13.8218,Z 60,A -33.5136,B 24.8429,C -2.8913,E1 25.1429,E2 -603.5139} C_DIS
LIN {X 28.0256,Y -15.7328,Z 60,A -36.8985,B 24.8435,C -2.8865,E1 25.1384,E2 -600.1352} C_DIS
LIN {X 27.0478,Y -17.36,Z 60,A -40.4846,B 24.8448,C -2.8744,E1 25.1331,E2 -596.5386} C_DIS
LIN {X 26.086,Y -18.7744,Z 60,A -43.1659,B 24.8451,C -2.8711,E1 25.1288,E2 -593.8626} C_DIS
LIN {X 25.0449,Y -20.1424,Z 60,A -46.9866,B 24.8471,C -2.8531,E1 25.1222,E2 -590.0173} C_DIS
LIN {X 23.0017,Y -22.4469,Z 60,A -51.78,B 24.8475,C -2.8488,E1 25.1131,E2 -585.2348} C_DIS
LIN {X 21.7425,Y -23.6688,Z 60,A -54.7202,B 24.848,C -2.844,E1 25.1072,E2 -582.2953} C_DIS
LIN {X 20.7778,Y -24.5195,Z 60,A -57.4236,B 24.8492,C -2.8337,E1 25.1014,E2 -579.5779} C_DIS
LIN {X 19.6299,Y -25.4483,Z 60,A -60.2652,B 24.85,C -2.8255,E1 25.0952,E2 -576.7274} C_DIS
LIN {X 17.9325,Y -26.6717,Z 60,A -63.4121,B 24.85,C -2.8255,E1 25.088,E2 -573.5913} C_DIS
LIN {X 16.5112,Y -27.5746,Z 60,A -66.6616,B 24.8509,C -2.8168,E1 25.0802,E2 -570.3317} C_DIS
LIN {X 14.8715,Y -28.4917,Z 60,A -69.9014,B 24.8514,C -2.8126,E1 25.0723,E2 -567.091} C_DIS
LIN {X 12.9889,Y -29.3982,Z 60,A -73.951,B 24.8524,C -2.803,E1 25.062,E2 -563.0289} C_DIS
LIN {X 11.2648,Y -30.1002,Z 60,A -76.7358,B 24.8522,C -2.8049,E1 25.0547,E2 -560.2549} C_DIS
LIN {X 9.8557,Y -30.5907,Z 60,A -79.6235,B 24.8528,C -2.799,E1 25.0471,E2 -557.3586} C_DIS
LIN {X 7.8541,Y -31.1647,Z 60,A -83.5946,B 24.8536,C -2.7921,E1 25.0363,E2 -553.3775} C_DIS
LIN {X 5.4947,Y -31.6662,Z 60,A -87.3055,B 24.8532,C -2.7953,E1 25.0262,E2 -549.6788} C_DIS
LIN {X 4.2567,Y -31.8562,Z 60,A -89.5663,B 24.8534,C -2.7935,E1 25.02,E2 -547.4156} C_DIS
LIN {X 2.9503,Y -32.0036,Z 60,A -92.0438,B 24.8537,C -2.7907,E1 25.0131,E2 -544.9331} C_DIS
LIN {X 1.3475,Y -32.111,Z 60,A -94.7433,B 24.8537,C -2.7914,E1 25.0055,E2 -542.2363} C_DIS
LIN {X 0.1197,Y -32.1384,Z 60,A -96.0087,B 24.8526,C -2.801,E1 25.0021,E2 -540.9938} C_DIS
Enddeposition()
LIN {X 0.1197,Y -32.1384,Z 60,A -96.0087,B 24.8526,C -2.801,E1 25.0021,E2 -540.9938} C_DIS
Startdeposition()
$VEL.CP = VEL_PRINT
LIN {X 1.0543,Y -31.1635,Z 60,A -93.7754,B 24.8502,C -2.8236,E1 25.0085,E2 -543.2805} C_DIS
LIN {X 3.3744,Y -30.998,Z 60,A -89.5002,B 24.85,C -2.8258,E1 25.0204,E2 -547.5584} C_DIS
LIN {X 5.5359,Y -30.6861,Z 60,A -85.3314,B 24.8495,C -2.8305,E1 25.0319,E2 -551.7342} C_DIS
LIN {X 7.684,Y -30.2194,Z 60,A -81.8831,B 24.8498,C -2.8274,E1 25.0412,E2 -555.1704} C_DIS
LIN {X 9.0101,Y -29.8513,Z 60,A -79.2571,B 24.8494,C -2.8313,E1 25.0483,E2 -557.8011} C_DIS
LIN {X 10.1777,Y -29.4734,Z 60,A -76.8788,B 24.849,C -2.8355,E1 25.0546,E2 -560.1848} C_DIS
LIN {X 11.6597,Y -28.9189,Z 60,A -73.9356,B 24.8485,C -2.8399,E1 25.0622,E2 -563.1318} C_DIS
LIN {X 13.3425,Y -28.1824,Z 60,A -70.3675,B 24.8477,C -2.8473,E1 25.0713,E2 -566.7085} C_DIS
LIN {X 15.6981,Y -26.9423,Z 60,A -65.1853,B 24.8464,C -2.8592,E1 25.084,E2 -571.904} C_DIS
LIN {X 17.8333,Y -25.5784,Z 60,A -61.1698,B 24.8464,C -2.8601,E1 25.0933,E2 -575.9082} C_DIS
LIN {X 19.2312,Y -24.545,Z 60,A -57.7676,B 24.8453,C -2.8694,E1 25.1009,E2 -579.32} C_DIS
LIN {X 20.5297,Y -23.4694,Z 60,A -55.0024,B 24.845,C -2.8719,E1 25.1067,E2 -582.0805} C_DIS
LIN {X 21.487,Y -22.5955,Z 60,A -52.4237,B 24.8442,C -2.88,E1 25.112,E2 -584.6677} C_DIS
LIN {X 22.8025,Y -21.2677,Z 60,A -49.0726,B 24.8434,C -2.8872,E1 25.1185,E2 -588.0213} C_DIS
LIN {X 23.9533,Y -19.9629,Z 60,A -45.8917,B 24.8425,C -2.895,E1 25.1243,E2 -591.2063} C_DIS
LIN {X 24.9987,Y -18.6374,Z 60,A -42.6484,B 24.8414,C -2.905,E1 25.1298,E2 -594.4579} C_DIS
LIN {X 26.2232,Y -16.8704,Z 60,A -39.0438,B 24.8408,C -2.9111,E1 25.1354,E2 -598.0592} C_DIS
LIN {X 27.2025,Y -15.2415,Z 60,A -35.1964,B 24.8392,C -2.9257,E1 25.1408,E2 -601.9213} C_DIS
LIN {X 28.1604,Y -13.3892,Z 60,A -31.4957,B 24.8381,C -2.935,E1 25.1454,E2 -605.6244} C_DIS
LIN {X 29.1727,Y -11.0089,Z 60,A -25.8485,B 24.8352,C -2.9615,E1 25.1513,E2 -611.3029} C_DIS
LIN {X 29.9671,Y -8.6178,Z 60,A -22.2384,B 24.8352,C -2.9615,E1 25.1542,E2 -614.8926} C_DIS
LIN {X 30.3516,Y -7.1441,Z 60,A -19.377,B 24.8341,C -2.9711,E1 25.1561,E2 -617.76} C_DIS
LIN {X 30.7297,Y -5.2897,Z 60,A -15.9973,B 24.833,C -2.9805,E1 25.1579,E2 -621.1423} C_DIS
LIN {X 30.987,Y -3.4768,Z 60,A -12.4884,B 24.8316,C -2.9931,E1 25.1591,E2 -624.6602} C_DIS
LIN {X 31.1456,Y -1.4774,Z 60,A -8.9261,B 24.8305,C -3.0029,E1 25.1597,E2 -628.2247} C_DIS
LIN {X 31.1787,Y 0.4322,Z 60,A -5.1764,B 24.8289,C -3.0172,E1 25.1597,E2 -631.9857} C_DIS
LIN {X 31.0092,Y 3.2713,Z 60,A 0.6137,B 24.8262,C -3.0411,E1 25.1583,E2 -637.7983} C_DIS
LIN {X 30.3685,Y 7.0725,Z 60,A 6.7788,B 24.8251,C -3.0499,E1 25.155,E2 -643.9483} C_DIS
LIN {X 29.8388,Y 9.0509,Z 60,A 10.1148,B 24.8245,C -3.0553,E1 25.1525,E2 -647.2777} C_DIS
LIN {X 29.4252,Y 10.316,Z 60,A 12.8631,B 24.8232,C -3.0664,E1 25.15,E2 -650.037} C_DIS
LIN {X 28.9382,Y 11.6118,Z 60,A 15.266,B 24.8226,C -3.0717,E1 25.1476,E2 -652.4391} C_DIS
LIN {X 28.385,Y 12.9065,Z 60,A 17.7697,B 24.8219,C -3.0778,E1 25.1448,E2 -654.9435} C_DIS
LIN {X 27.7748,Y 14.1718,Z 60,A 20.7476,B 24.8205,C -3.09,E1 25.141,E2 -657.9345} C_DIS
LIN {X 26.5119,Y 16.4138,Z 60,A 25.7099,B 24.8187,C -3.1053,E1 25.134,E2 -662.9077} C_DIS
LIN {X 25.2414,Y 18.3073,Z 60,A 29.6533,B 24.8179,C -3.1123,E1 25.1276,E2 -666.8483} C_DIS
LIN {X 23.6004,Y 20.379,Z 60,A 33.8746,B 24.8175,C -3.1153,E1 25.1202,E2 -671.0572} C_DIS
LIN {X 22.3378,Y 21.7556,Z 60,A 38.303,B 24.8152,C -3.1352,E1 25.1116,E2 -675.5137} C_DIS
LIN {X 20.7346,Y 23.2887,Z 60,A 41.897,B 24.8149,C -3.1372,E1 25.1043,E2 -679.0977} C_DIS
LIN {X 19.0515,Y 24.6845,Z 60,A 45.5264,B 24.8147,C -3.1396,E1 25.0964,E2 -682.7192} C_DIS
LIN {X 17.7132,Y 25.6612,Z 60,A 49.0782,B 24.8133,C -3.1508,E1 25.0883,E2 -686.2853} C_DIS
LIN {X 15.5118,Y 27.0493,Z 60,A 53.4233,B 24.8131,C -3.1525,E1 25.0779,E2 -690.6208} C_DIS
LIN {X 13.6406,Y 28.039,Z 60,A 57.9888,B 24.8116,C -3.1652,E1 25.0665,E2 -695.2041} C_DIS
LIN {X 11.3068,Y 29.0588,Z 60,A 62.0159,B 24.8119,C -3.1624,E1 25.0561,E2 -699.2153} C_DIS
LIN {X 9.4932,Y 29.7007,Z 60,A 65.6301,B 24.8115,C -3.1662,E1 25.0466,E2 -702.8314} C_DIS
LIN {X 7.6891,Y 30.2181,Z 60,A 68.9931,B 24.8113,C -3.1674,E1 25.0375,E2 -706.192} C_DIS
LIN {X 5.8076,Y 30.6355,Z 60,A 72.6037,B 24.8111,C -3.1697,E1 25.0276,E2 -709.8035} C_DIS
LIN {X 3.9305,Y 30.9327,Z 60,A 75.7558,B 24.8114,C -3.167,E1 25.019,E2 -712.9463} C_DIS
LIN {X 2.8125,Y 31.0543,Z 60,A 77.9312,B 24.8112,C -3.1684,E1 25.0129,E2 -715.1237} C_DIS
LIN {X 1.5034,Y 31.1447,Z 60,A 80.4289,B 24.8112,C -3.1692,E1 25.0059,E2 -717.6224} C_DIS
LIN {X -0.1002,Y 31.1809,Z 60,A 83.4801,B 24.8111,C -3.1698,E1 24.9974,E2 -720.6748} C_DIS
LIN {X -1.8789,Y 31.1243,Z 60,A 86.8709,B 24.8111,C -3.1699,E1 24.988,E2 -724.0666} C_DIS
LIN {X -4.0272,Y 30.9201,Z 60,A 90.6106,B 24.8116,C -3.1656,E1 24.9776,E2 -727.7982} C_DIS
LIN {X -5.5559,Y 30.682,Z 60,A 93.8473,B 24.8113,C -3.1674,E1 24.9687,E2 -731.0424} C_DIS
LIN {X -7.7892,Y 30.1922,Z 60,A 97.8112,B 24.8121,C -3.1613,E1 24.9579,E2 -734.9971} C_DIS
LIN {X -9.6775,Y 29.6415,Z 60,A 101.1922,B 24.8128,C -3.1552,E1 24.9489,E2 -738.3693} C_DIS
LIN {X -10.8512,Y 29.2319,Z 60,A 103.7873,B 24.8128,C -3.1552,E1 24.9421,E2 -740.9696} C_DIS
LIN {X -12.7741,Y 28.4444,Z 60,A 107.6457,B 24.8134,C -3.1501,E1 24.9322,E2 -744.825} C_DIS
LIN {X -14.6236,Y 27.5397,Z 60,A 111.1018,B 24.8145,C -3.1413,E1 24.9236,E2 -748.2692} C_DIS
LIN {X -16.0654,Y 26.7246,Z 60,A 114.4539,B 24.8148,C -3.1386,E1 24.9155,E2 -751.625} C_DIS
LIN {X -17.4051,Y 25.8715,Z 60,A 117.5237,B 24.8153,C -3.1345,E1 24.9084,E2 -754.6949} C_DIS
LIN {X -18.6835,Y 24.9641,Z 60,A 120.6562,B 24.8157,C -3.1308,E1 24.9013,E2 -757.8298} C_DIS
LIN {X -20.0124,Y 23.9121,Z 60,A 123.5953,B 24.8167,C -3.1227,E1 24.895,E2 -760.7607} C_DIS
LIN {X -21.6986,Y 22.3929,Z 60,A 127.9599,B 24.8176,C -3.1148,E1 24.8862,E2 -765.1243} C_DIS
LIN {X -23.5756,Y 20.4075,Z 60,A 132.2817,B 24.8197,C -3.097,E1 24.878,E2 -769.4226} C_DIS
LIN {X -24.3244,Y 19.5097,Z 60,A 134.6193,B 24.8201,C -3.093,E1 24.8739,E2 -771.7615} C_DIS
LIN {X -25.1742,Y 18.3991,Z 60,A 137.4932,B 24.8207,C -3.0886,E1 24.8691,E2 -774.6389} C_DIS
LIN {X -26.3057,Y 16.7417,Z 60,A 141.9609,B 24.8211,C -3.0847,E1 24.8623,E2 -779.1195} C_DIS
LIN {X -28.2686,Y 13.1585,Z 60,A 148.3078,B 24.8246,C -3.0543,E1 24.8542,E2 -785.4277} C_DIS
LIN {X -29.1071,Y 11.1808,Z 60,A 152.959,B 24.8254,C -3.0479,E1 24.8493,E2 -790.0893} C_DIS
LIN {X -29.8699,Y 8.9463,Z 60,A 157.2034,B 24.827,C -3.034,E1 24.8457,E2 -794.3248} C_DIS
LIN {X -30.3998,Y 6.9375,Z 60,A 160.9072,B 24.8284,C -3.0214,E1 24.8432,E2 -798.0202} C_DIS
LIN {X -30.7875,Y 4.9421,Z 60,A 164.6357,B 24.8297,C -3.0098,E1 24.8414,E2 -801.7429} C_DIS
LIN {X -31.0289,Y 3.0736,Z 60,A 168.4516,B 24.8307,C -3.0016,E1 24.8403,E2 -805.562} C_DIS
LIN {X -31.1766,Y 0.523,Z 60,A 173.4313,B 24.8321,C -2.989,E1 24.8398,E2 -810.5415} C_DIS
LIN {X -31.0598,Y -2.7524,Z 60,A 178.9441,B 24.8346,C -2.9665,E1 24.8407,E2 -816.0337} C_DIS
LIN {X -30.9108,Y -4.098,Z 60,A -178.6961,B 24.8356,C -2.958,E1 24.8415,E2 -818.387} C_DIS
LIN {X -30.6595,Y -5.6797,Z 60,A -175.9197,B 24.8367,C -2.9478,E1 24.8428,E2 -821.1556} C_DIS
LIN {X -30.2855,Y -7.4204,Z 60,A -172.4933,B 24.8377,C -2.9391,E1 24.8449,E2 -824.5814} C_DIS
LIN {X -29.5749,Y -9.878,Z 60,A -167.3676,B 24.8388,C -2.9286,E1 24.8491,E2 -829.7115} C_DIS
LIN {X -28.8495,Y -11.8311,Z 60,A -163.7196,B 24.8402,C -2.9164,E1 24.8528,E2 -833.3506} C_DIS
LIN {X -27.9126,Y -13.8982,Z 60,A -159.0014,B 24.841,C -2.9093,E1 24.8585,E2 -838.0775} C_DIS
LIN {X -26.1899,Y -16.9215,Z 60,A -152.6486,B 24.8428,C -2.8926,E1 24.8676,E2 -844.423} C_DIS
LIN {X -24.6366,Y -19.1131,Z 60,A -147.6997,B 24.8441,C -2.881,E1 24.8759,E2 -849.3679} C_DIS
LIN {X -23.1564,Y -20.8824,Z 60,A -143.8166,B 24.8454,C -2.8686,E1 24.883,E2 -853.239} C_DIS
LIN {X -21.5793,Y -22.5082,Z 60,A -139.481,B 24.8461,C -2.8616,E1 24.8916,E2 -857.5761} C_DIS
LIN {X -20.1344,Y -23.8097,Z 60,A -136.2421,B 24.8472,C -2.852,E1 24.8984,E2 -860.8047} C_DIS
LIN {X -18.7167,Y -24.9392,Z 60,A -132.7698,B 24.8477,C -2.8474,E1 24.906,E2 -864.2789} C_DIS
LIN {X -16.6708,Y -26.3504,Z 60,A -127.4414,B 24.8477,C -2.8474,E1 24.9185,E2 -869.6246} C_DIS
LIN {X -14.5491,Y -27.5788,Z 60,A -123.4787,B 24.8489,C -2.8364,E1 24.9282,E2 -873.5724} C_DIS
LIN {X -12.5599,Y -28.5402,Z 60,A -119.4427,B 24.8494,C -2.8317,E1 24.9384,E2 -877.6073} C_DIS
LIN {X -10.1755,Y -29.4741,Z 60,A -114.3827,B 24.8494,C -2.8311,E1 24.9517,E2 -882.6761} C_DIS
LIN {X -7.8468,Y -30.178,Z 60,A -109.6664,B 24.8494,C -2.8309,E1 24.9644,E2 -887.3991} C_DIS
LIN {X -4.3589,Y -30.8752,Z 60,A -103.6998,B 24.8503,C -2.8229,E1 24.9808,E2 -893.3527} C_DIS
LIN {X -2.231,Y -31.1011,Z 60,A -99.9597,B 24.8505,C -2.8207,E1 24.9912,E2 -897.0893} C_DIS
LIN {X -0.1621,Y -31.181,Z 60,A -95.8698,B 24.8501,C -2.8244,E1 25.0026,E2 -901.1883} C_DIS
LIN {X -0.1621,Y -31.181,Z 60,A -95.8698,B 24.8501,C -2.8244,E1 25.0026,E2 -901.1883} C_DIS
Enddeposition()
LIN {X 0.0842,Y -30.2228,Z 60,A -95.4358,B 24.8484,C -2.8405,E1 25.0039,E2 -901.6607} C_DIS
Startdeposition()
$VEL.CP = VEL_PRINT
LIN {X -1.136,Y -30.2018,Z 60,A -99.4718,B 24.8504,C -2.8222,E1 24.9925,E2 -897.5811} C_DIS
LIN {X -2.8098,Y -30.0921,Z 60,A -102.9498,B 24.8507,C -2.8193,E1 24.9828,E2 -894.0947} C_DIS
LIN {X -4.5561,Y -29.878,Z 60,A -106.5578,B 24.8509,C -2.8174,E1 24.9728,E2 -890.4791} C_DIS
LIN {X -7.0476,Y -29.3896,Z 60,A -111.0812,B 24.8504,C -2.8222,E1 24.9605,E2 -885.9617} C_DIS
LIN {X -8.9602,Y -28.8643,Z 60,A -114.8683,B 24.8501,C -2.8244,E1 24.9504,E2 -882.1737} C_DIS
LIN {X -10.8145,Y -28.2224,Z 60,A -118.4393,B 24.8497,C -2.829,E1 24.941,E2 -878.6063} C_DIS
LIN {X -12.6326,Y -27.4562,Z 60,A -122.3559,B 24.8494,C -2.8313,E1 24.931,E2 -874.686} C_DIS
LIN {X -14.2006,Y -26.6795,Z 60,A -125.5468,B 24.8488,C -2.8365,E1 24.9231,E2 -871.4988} C_DIS
LIN {X -16.183,Y -25.5254,Z 60,A -130.3199,B 24.8486,C -2.8391,E1 24.9116,E2 -866.7172} C_DIS
LIN {X -18.1911,Y -24.1357,Z 60,A -134.9649,B 24.8478,C -2.8466,E1 24.9011,E2 -862.0738} C_DIS
LIN {X -20.0135,Y -22.6475,Z 60,A -139.6219,B 24.847,C -2.8533,E1 24.8912,E2 -857.4148} C_DIS
LIN {X -22.2078,Y -20.5002,Z 60,A -144.9277,B 24.8453,C -2.8694,E1 24.8809,E2 -852.1248} C_DIS
LIN {X -23.8307,Y -18.5883,Z 60,A -150.171,B 24.8445,C -2.8765,E1 24.8716,E2 -846.8742} C_DIS
LIN {X -25.2447,Y -16.6179,Z 60,A -154.5729,B 24.8432,C -2.8892,E1 24.8647,E2 -842.481} C_DIS
LIN {X -26.2059,Y -15.0564,Z 60,A -157.6624,B 24.8419,C -2.901,E1 24.8603,E2 -839.4037} C_DIS
LIN {X -27.0416,Y -13.4981,Z 60,A -161.3723,B 24.8412,C -2.9074,E1 24.8555,E2 -835.6892} C_DIS
LIN {X -27.8012,Y -11.8547,Z 60,A -164.6191,B 24.84,C -2.9182,E1 24.8518,E2 -832.4504} C_DIS
LIN {X -28.3363,Y -10.5108,Z 60,A -167.1608,B 24.839,C -2.9274,E1 24.8493,E2 -829.9164} C_DIS
LIN {X -28.8891,Y -8.8799,Z 60,A -171.0566,B 24.8384,C -2.9325,E1 24.8459,E2 -826.0105} C_DIS
LIN {X -29.5248,Y -6.4595,Z 60,A -175.442,B 24.8366,C -2.9491,E1 24.843,E2 -821.6392} C_DIS
LIN {X -29.8206,Y -4.9169,Z 60,A -178.3851,B 24.8355,C -2.9583,E1 24.8416,E2 -818.7008} C_DIS
LIN {X -30.0647,Y -3.0914,Z 60,A 177.2752,B 24.835,C -2.9634,E1 24.8402,E2 -814.3472} C_DIS
LIN {X -30.2214,Y -0.0752,Z 60,A 172.7618,B 24.832,C -2.9893,E1 24.8398,E2 -809.8688} C_DIS
LIN {X -30.1948,Y 1.3077,Z 60,A 169.0114,B 24.832,C -2.9899,E1 24.8401,E2 -806.0973} C_DIS
LIN {X -29.9492,Y 4.062,Z 60,A 164.09,B 24.8299,C -3.0084,E1 24.8417,E2 -801.1907} C_DIS
LIN {X -29.633,Y 5.9431,Z 60,A 160.3925,B 24.8287,C -3.0191,E1 24.8435,E2 -797.4969} C_DIS
LIN {X -28.9492,Y 8.6797,Z 60,A 154.9013,B 24.8269,C -3.0346,E1 24.8476,E2 -792.0107} C_DIS
LIN {X -28.1579,Y 10.9796,Z 60,A 150.2227,B 24.8254,C -3.0479,E1 24.8521,E2 -787.3377} C_DIS
LIN {X -27.1801,Y 13.2171,Z 60,A 145.6023,B 24.8238,C -3.0615,E1 24.8575,E2 -782.7245} C_DIS
LIN {X -26.0167,Y 15.3801,Z 60,A 141.5271,B 24.8218,C -3.0786,E1 24.863,E2 -778.6691} C_DIS
LIN {X -25.2748,Y 16.5722,Z 60,A 138.8534,B 24.821,C -3.0858,E1 24.867,E2 -775.999} C_DIS
LIN {X -24.2739,Y 18.0062,Z 60,A 135.1264,B 24.8203,C -3.0917,E1 24.8731,E2 -772.2678} C_DIS
LIN {X -23.0798,Y 19.5134,Z 60,A 131.5244,B 24.8192,C -3.1012,E1 24.8794,E2 -768.672} C_DIS
LIN {X -21.988,Y 20.7359,Z 60,A 128.634,B 24.8181,C -3.1104,E1 24.8849,E2 -765.7907} C_DIS
LIN {X -20.8918,Y 21.8401,Z 60,A 125.454,B 24.8175,C -3.1155,E1 24.8912,E2 -762.6097} C_DIS
LIN {X -19.7021,Y 22.9189,Z 60,A 122.2086,B 24.8169,C -3.1207,E1 24.898,E2 -759.3639} C_DIS
LIN {X -18.2782,Y 24.0703,Z 60,A 119.249,B 24.8156,C -3.1318,E1 24.9045,E2 -756.42} C_DIS
LIN {X -16.9774,Y 25.0043,Z 60,A 115.8205,B 24.8152,C -3.1347,E1 24.9123,E2 -752.9866} C_DIS
LIN {X -15.627,Y 25.8699,Z 60,A 113.006,B 24.8144,C -3.142,E1 24.919,E2 -750.1807} C_DIS
LIN {X -13.9905,Y 26.7899,Z 60,A 109.0967,B 24.814,C -3.145,E1 24.9286,E2 -746.2676} C_DIS
LIN {X -12.0096,Y 27.7343,Z 60,A 104.9928,B 24.8132,C -3.1516,E1 24.939,E2 -742.1694} C_DIS
LIN {X -10.0711,Y 28.4957,Z 60,A 100.8711,B 24.8128,C -3.1552,E1 24.9498,E2 -738.0476} C_DIS
LIN {X -7.9984,Y 29.1454,Z 60,A 97.2271,B 24.8118,C -3.1637,E1 24.9595,E2 -734.418} C_DIS
LIN {X -6.8088,Y 29.446,Z 60,A 94.6387,B 24.8118,C -3.1635,E1 24.9665,E2 -731.8255} C_DIS
LIN {X -4.996,Y 29.8075,Z 60,A 91.1946,B 24.8114,C -3.1667,E1 24.976,E2 -728.3854} C_DIS
LIN {X -3.2246,Y 30.0506,Z 60,A 88.0819,B 24.8109,C -3.1712,E1 24.9846,E2 -725.2813} C_DIS
LIN {X -2.0657,Y 30.1526,Z 60,A 85.439,B 24.8113,C -3.1681,E1 24.992,E2 -722.6297} C_DIS
LIN {X 0.3609,Y 30.2212,Z 60,A 80.5263,B 24.8115,C -3.1661,E1 25.0057,E2 -717.7124} C_DIS
LIN {X 2.5708,Y 30.1134,Z 60,A 76.4205,B 24.8115,C -3.1669,E1 25.0171,E2 -713.6102} C_DIS
LIN {X 5.0311,Y 29.8016,Z 60,A 71.9454,B 24.8113,C -3.1679,E1 25.0295,E2 -709.1417} C_DIS
LIN {X 6.649,Y 29.483,Z 60,A 68.6381,B 24.8117,C -3.1646,E1 25.0385,E2 -705.8307} C_DIS
LIN {X 8.3978,Y 29.033,Z 60,A 65.3789,B 24.8117,C -3.1641,E1 25.0473,E2 -702.5758} C_DIS
LIN {X 10.3457,Y 28.3971,Z 60,A 61.3547,B 24.8123,C -3.1594,E1 25.0579,E2 -698.5483} C_DIS
LIN {X 11.7628,Y 27.8402,Z 60,A 58.3493,B 24.8128,C -3.1551,E1 25.0656,E2 -695.5398} C_DIS
LIN {X 13.8859,Y 26.8444,Z 60,A 54.3875,B 24.8128,C -3.1551,E1 25.0755,E2 -691.5886} C_DIS
LIN {X 15.4376,Y 25.9832,Z 60,A 50.4123,B 24.8142,C -3.1436,E1 25.0852,E2 -687.5979} C_DIS
LIN {X 17.8013,Y 24.4247,Z 60,A 45.5962,B 24.8145,C -3.1413,E1 25.0962,E2 -682.7928} C_DIS
LIN {X 19.3503,Y 23.2164,Z 60,A 42.2499,B 24.8147,C -3.139,E1 25.1035,E2 -679.4537} C_DIS
LIN {X 20.4931,Y 22.2146,Z 60,A 38.9885,B 24.8159,C -3.129,E1 25.1103,E2 -676.1814} C_DIS
LIN {X 21.7018,Y 21.0348,Z 60,A 35.9084,B 24.8165,C -3.1238,E1 25.1164,E2 -673.1021} C_DIS
LIN {X 23.1192,Y 19.4669,Z 60,A 31.5658,B 24.8181,C -3.1108,E1 25.1244,E2 -668.7484} C_DIS
LIN {X 24.394,Y 17.8433,Z 60,A 28.2601,B 24.8183,C -3.109,E1 25.1299,E2 -665.4541} C_DIS
LIN {X 25.0435,Y 16.9194,Z 60,A 25.1815,B 24.8202,C -3.0922,E1 25.1348,E2 -662.3508} C_DIS
LIN {X 26.7959,Y 13.9791,Z 60,A 19.8922,B 24.8205,C -3.0903,E1 25.1421,E2 -657.0843} C_DIS
LIN {X 27.5316,Y 12.468,Z 60,A 15.9953,B 24.8225,C -3.0726,E1 25.1468,E2 -653.1664} C_DIS
LIN {X 28.3661,Y 10.4305,Z 60,A 12.3221,B 24.8232,C -3.0671,E1 25.1505,E2 -649.5008} C_DIS
LIN {X 28.7927,Y 9.1866,Z 60,A 9.7451,B 24.8241,C -3.0588,E1 25.1528,E2 -646.9187} C_DIS
LIN {X 29.2327,Y 7.6734,Z 60,A 6.4783,B 24.8255,C -3.0464,E1 25.1552,E2 -643.6411} C_DIS
LIN {X 29.8039,Y 5.0178,Z 60,A 0.8164,B 24.8281,C -3.0242,E1 25.1582,E2 -637.9598} C_DIS
LIN {X 30.127,Y 2.4011,Z 60,A -3.6581,B 24.8291,C -3.0156,E1 25.1595,E2 -633.4913} C_DIS
LIN {X 30.2216,Y 0.2532,Z 60,A -7.7988,B 24.8306,C -3.002,E1 25.1598,E2 -629.3431} C_DIS
LIN {X 30.1128,Y -2.5791,Z 60,A -13.5455,B 24.8331,C -2.9804,E1 25.1588,E2 -623.5792} C_DIS
LIN {X 29.7211,Y -5.486,Z 60,A -18.8131,B 24.8346,C -2.9668,E1 25.1564,E2 -618.3106} C_DIS
LIN {X 29.0187,Y -8.4471,Z 60,A -25.3256,B 24.8376,C -2.9395,E1 25.1517,E2 -611.7709} C_DIS
LIN {X 27.5831,Y -12.3533,Z 60,A -31.6783,B 24.838,C -2.9358,E1 25.1452,E2 -605.4446} C_DIS
LIN {X 27.0077,Y -13.5659,Z 60,A -34.551,B 24.8393,C -2.9242,E1 25.1417,E2 -602.5598} C_DIS
LIN {X 25.9938,Y -15.4194,Z 60,A -38.3416,B 24.8403,C -2.9156,E1 25.1365,E2 -598.7685} C_DIS
LIN {X 24.9647,Y -17.0358,Z 60,A -42.2489,B 24.8417,C -2.9022,E1 25.1304,E2 -594.8489} C_DIS
LIN {X 23.5344,Y -18.9627,Z 60,A -46.7226,B 24.8429,C -2.8913,E1 25.1228,E2 -590.3705} C_DIS
LIN {X 22.2937,Y -20.4068,Z 60,A -50.2983,B 24.8439,C -2.8827,E1 25.1162,E2 -586.7905} C_DIS
LIN {X 20.949,Y -21.785,Z 60,A -53.753,B 24.8445,C -2.8765,E1 25.1093,E2 -583.3357} C_DIS
LIN {X 19.8619,Y -22.7805,Z 60,A -56.4303,B 24.8451,C -2.8717,E1 25.1037,E2 -580.6576} C_DIS
LIN {X 18.3759,Y -23.9954,Z 60,A -60.1015,B 24.8459,C -2.8636,E1 25.0957,E2 -576.9808} C_DIS
LIN {X 17.1329,Y -24.8982,Z 60,A -63.2324,B 24.8468,C -2.8552,E1 25.0885,E2 -573.8408} C_DIS
LIN {X 15.3155,Y -26.0555,Z 60,A -67.3394,B 24.8477,C -2.8474,E1 25.0788,E2 -569.7285} C_DIS
LIN {X 13.4645,Y -27.0582,Z 60,A -71.2129,B 24.8482,C -2.8422,E1 25.0692,E2 -565.8534} C_DIS
LIN {X 12.0463,Y -27.7184,Z 60,A -73.7949,B 24.8482,C -2.8422,E1 25.0626,E2 -563.2778} C_DIS
LIN {X 10.6661,Y -28.2782,Z 60,A -76.9533,B 24.849,C -2.8346,E1 25.0544,E2 -560.1083} C_DIS
LIN {X 8.85,Y -28.8982,Z 60,A -80.4709,B 24.8494,C -2.8317,E1 25.045,E2 -556.5904} C_DIS
LIN {X 7.3092,Y -29.326,Z 60,A -84.1164,B 24.8504,C -2.8219,E1 25.0351,E2 -552.9272} C_DIS
LIN {X 4.6552,Y -29.8627,Z 60,A -88.9482,B 24.8504,C -2.8211,E1 25.0218,E2 -548.0989} C_DIS
LIN {X 2.0803,Y -30.1513,Z 60,A -93.5104,B 24.8504,C -2.8223,E1 25.0092,E2 -543.5421} C_DIS
LIN {X 0.0842,Y -30.2228,Z 60,A -95.4357,B 24.8484,C -2.8405,E1 25.004,E2 -541.6607} C_DIS
Enddeposition()
LIN {X 0.0842,Y -30.2228,Z 60,A -95.4357,B 24.8484,C -2.8405,E1 25.004,E2 -541.6607} C_DIS
Startdeposition()
$VEL.CP = VEL_PRINT
LIN {X 0.4198,Y -29.2621,Z 60,A -95.1938,B 24.8471,C -2.8526,E1 25.0047,E2 -541.9314} C_DIS
LIN {X 1.9172,Y -29.2022,Z 60,A -92.3979,B 24.8471,C -2.8524,E1 25.0125,E2 -544.7257} C_DIS
LIN {X 3.1517,Y -29.0943,Z 60,A -89.7748,B 24.8468,C -2.8557,E1 25.0198,E2 -547.3552} C_DIS
LIN {X 4.8557,Y -28.8595,Z 60,A -86.3921,B 24.8465,C -2.8582,E1 25.0291,E2 -550.7407} C_DIS
LIN {X 6.5646,Y -28.5193,Z 60,A -83.1438,B 24.8464,C -2.8594,E1 25.038,E2 -553.9876} C_DIS
LIN {X 7.8597,Y -28.1895,Z 60,A -80.5526,B 24.8461,C -2.8619,E1 25.045,E2 -556.5805} C_DIS
LIN {X 9.2753,Y -27.756,Z 60,A -77.1264,B 24.8451,C -2.8712,E1 25.0541,E2 -560.0224} C_DIS
LIN {X 11.3125,Y -26.99,Z 60,A -73.5129,B 24.8453,C -2.8696,E1 25.0635,E2 -563.6242} C_DIS
LIN {X 12.7626,Y -26.3352,Z 60,A -70.1769,B 24.8445,C -2.8769,E1 25.072,E2 -566.9689} C_DIS
LIN {X 14.2261,Y -25.5748,Z 60,A -67.2469,B 24.8443,C -2.8788,E1 25.0792,E2 -569.8952} C_DIS
LIN {X 15.1443,Y -25.042,Z 60,A -64.8959,B 24.8435,C -2.8857,E1 25.0848,E2 -572.2554} C_DIS
LIN {X 16.4313,Y -24.217,Z 60,A -61.7992,B 24.8428,C -2.8927,E1 25.092,E2 -575.3583} C_DIS
LIN {X 18.0112,Y -23.0658,Z 60,A -58.3313,B 24.8424,C -2.8963,E1 25.0998,E2 -578.8222} C_DIS
LIN {X 18.8644,Y -22.374,Z 60,A -54.8268,B 24.8401,C -2.9175,E1 25.1073,E2 -582.3634} C_DIS
LIN {X 21.7341,Y -19.598,Z 60,A -47.9787,B 24.8393,C -2.9241,E1 25.1207,E2 -589.1978} C_DIS
LIN {X 23.0643,Y -18.0137,Z 60,A -44.0254,B 24.8383,C -2.9332,E1 25.1276,E2 -593.1545} C_DIS
LIN {X 24.0737,Y -16.6406,Z 60,A -40.8084,B 24.8375,C -2.9407,E1 25.1329,E2 -596.3734} C_DIS
LIN {X 25.049,Y -15.1328,Z 60,A -37.4252,B 24.8366,C -2.9487,E1 25.1379,E2 -599.7585} C_DIS
LIN {X 25.7535,Y -13.8992,Z 60,A -34.8466,B 24.836,C -2.954,E1 25.1414,E2 -602.3362} C_DIS
LIN {X 26.2966,Y -12.8418,Z 60,A -32.3532,B 24.835,C -2.9629,E1 25.1445,E2 -604.8374} C_DIS
LIN {X 27.1054,Y -11.0333,Z 60,A -28.0351,B 24.8331,C -2.98,E1 25.1493,E2 -609.1724} C_DIS
LIN {X 27.7367,Y -9.333,Z 60,A -24.9868,B 24.8326,C -2.9842,E1 25.1521,E2 -612.2135} C_DIS
LIN {X 28.2246,Y -7.7337,Z 60,A -21.356,B 24.831,C -2.9989,E1 25.1549,E2 -615.8583} C_DIS
LIN {X 28.7078,Y -5.6831,Z 60,A -17.3595,B 24.8297,C -3.01,E1 25.1573,E2 -619.8578} C_DIS
LIN {X 29.0492,Y -3.5456,Z 60,A -13.3657,B 24.8286,C -3.02,E1 25.1588,E2 -623.8519} C_DIS
LIN {X 29.2047,Y -1.8758,Z 60,A -9.8962,B 24.8271,C -3.0327,E1 25.1596,E2 -627.3309} C_DIS
LIN {X 29.2635,Y 0.074,Z 60,A -6.4767,B 24.8263,C -3.0395,E1 25.1598,E2 -630.7461} C_DIS
LIN {X 29.2255,Y 1.5116,Z 60,A -3.2685,B 24.8247,C -3.0533,E1 25.1594,E2 -633.968} C_DIS
LIN {X 29.0474,Y 3.5622,Z 60,A 0.838,B 24.8232,C -3.0668,E1 25.1582,E2 -638.082} C_DIS
LIN {X 28.674,Y 5.8509,Z 60,A 5.1666,B 24.8219,C -3.0778,E1 25.156,E2 -642.4114} C_DIS
LIN {X 28.1852,Y 7.8751,Z 60,A 8.4895,B 24.8216,C -3.0803,E1 25.1538,E2 -645.7209} C_DIS
LIN {X 27.6144,Y 9.689,Z 60,A 12.7525,B 24.8196,C -3.0979,E1 25.1501,E2 -650.0017} C_DIS
LIN {X 27.0253,Y 11.2282,Z 60,A 15.605,B 24.8191,C -3.1023,E1 25.1471,E2 -652.8488} C_DIS
LIN {X 26.4507,Y 12.5229,Z 60,A 18.6297,B 24.8178,C -3.1131,E1 25.1436,E2 -655.8826} C_DIS
LIN {X 25.8104,Y 13.7948,Z 60,A 22.1362,B 24.8158,C -3.1296,E1 25.139,E2 -659.4096} C_DIS
LIN {X 24.3493,Y 16.2345,Z 60,A 26.9005,B 24.8154,C -3.1337,E1 25.132,E2 -664.1596} C_DIS
LIN {X 23.5463,Y 17.3791,Z 60,A 29.9776,B 24.8141,C -3.1445,E1 25.127,E2 -667.2474} C_DIS
LIN {X 22.5619,Y 18.6392,Z 60,A 32.6052,B 24.8139,C -3.1456,E1 25.1224,E2 -669.8654} C_DIS
LIN {X 21.1968,Y 20.1778,Z 60,A 37.7375,B 24.8113,C -3.1676,E1 25.1126,E2 -675.0273} C_DIS
LIN {X 19.6643,Y 21.6742,Z 60,A 42.0446,B 24.8102,C -3.1772,E1 25.1038,E2 -679.3397} C_DIS
LIN {X 17.1099,Y 23.7426,Z 60,A 47.9814,B 24.8095,C -3.1825,E1 25.0906,E2 -685.2675} C_DIS
LIN {X 14.7233,Y 25.2923,Z 60,A 52.977,B 24.8093,C -3.1843,E1 25.0788,E2 -690.2513} C_DIS
LIN {X 12.9502,Y 26.2435,Z 60,A 57.3301,B 24.8082,C -3.1938,E1 25.068,E2 -694.6151} C_DIS
LIN {X 11.3077,Y 26.992,Z 60,A 60.2945,B 24.8085,C -3.1914,E1 25.0604,E2 -697.5665} C_DIS
LIN {X 9.9836,Y 27.5092,Z 60,A 63.29,B 24.8079,C -3.1962,E1 25.0526,E2 -700.5671} C_DIS
LIN {X 8.2439,Y 28.0797,Z 60,A 67.0317,B 24.8074,C -3.2005,E1 25.0426,E2 -704.3123} C_DIS
LIN {X 6.2106,Y 28.5983,Z 60,A 71.0544,B 24.8072,C -3.2018,E1 25.0317,E2 -708.3323} C_DIS
LIN {X 4.0423,Y 28.9847,Z 60,A 75.7179,B 24.8066,C -3.2066,E1 25.0188,E2 -713.0028} C_DIS
LIN {X 1.8873,Y 29.204,Z 60,A 80.5564,B 24.8059,C -3.2127,E1 25.0053,E2 -717.8535} C_DIS
LIN {X -2.2529,Y 29.1781,Z 60,A 88.5163,B 24.8064,C -3.2087,E1 24.9831,E2 -725.8053} C_DIS
LIN {X -5.1974,Y 28.7999,Z 60,A 94.0104,B 24.8072,C -3.2019,E1 24.968,E2 -731.288} C_DIS
LIN {X -8.1725,Y 28.1007,Z 60,A 98.8717,B 24.8091,C -3.1864,E1 24.9549,E2 -736.1191} C_DIS
LIN {X -9.8561,Y 27.5549,Z 60,A 103.3261,B 24.8085,C -3.1907,E1 24.9431,E2 -740.5924} C_DIS
LIN {X -12.0268,Y 26.6793,Z 60,A 108.1503,B 24.8091,C -3.1863,E1 24.9307,E2 -745.4172} C_DIS
LIN {X -14.4521,Y 25.4477,Z 60,A 112.6545,B 24.8109,C -3.1709,E1 24.9197,E2 -749.8972} C_DIS
LIN {X -15.4574,Y 24.85,Z 60,A 115.3706,B 24.811,C -3.1702,E1 24.9132,E2 -752.6201} C_DIS
LIN {X -17.2416,Y 23.6469,Z 60,A 119.0139,B 24.8125,C -3.1576,E1 24.9049,E2 -756.2456} C_DIS
LIN {X -18.5777,Y 22.6129,Z 60,A 122.9565,B 24.8128,C -3.1555,E1 24.8962,E2 -760.1979} C_DIS
LIN {X -20.4349,Y 20.9496,Z 60,A 128.0583,B 24.8139,C -3.1461,E1 24.8858,E2 -765.298} C_DIS
LIN {X -21.6739,Y 19.6645,Z 60,A 131.3876,B 24.815,C -3.1364,E1 24.8795,E2 -768.6187} C_DIS
LIN {X -22.9584,Y 18.1484,Z 60,A 135.1025,B 24.8164,C -3.1253,E1 24.873,E2 -772.3242} C_DIS
LIN {X -24.0609,Y 16.6587,Z 60,A 138.5662,B 24.8176,C -3.1145,E1 24.8673,E2 -775.7791} C_DIS
LIN {X -25.2744,Y 14.7536,Z 60,A 143.8239,B 24.8184,C -3.1081,E1 24.8597,E2 -781.0485} C_DIS
LIN {X -26.2499,Y 12.9373,Z 60,A 147.0604,B 24.8204,C -3.091,E1 24.8556,E2 -784.2613} C_DIS
LIN {X -26.9013,Y 11.5216,Z 60,A 150.5523,B 24.8211,C -3.0851,E1 24.8516,E2 -787.7582} C_DIS
LIN {X -27.6383,Y 9.6204,Z 60,A 154.6387,B 24.8224,C -3.0738,E1 24.8477,E2 -791.8406} C_DIS
LIN {X -28.3339,Y 7.3227,Z 60,A 159.253,B 24.8241,C -3.0588,E1 24.8442,E2 -796.4459} C_DIS
LIN {X -28.7787,Y 5.3142,Z 60,A 163.2415,B 24.8256,C -3.0461,E1 24.842,E2 -800.4274} C_DIS
LIN {X -29.0565,Y 3.4867,Z 60,A 166.9414,B 24.8268,C -3.0354,E1 24.8406,E2 -804.1237} C_DIS
LIN {X -29.1934,Y 2.0444,Z 60,A 169.4083,B 24.8281,C -3.0241,E1 24.8401,E2 -806.5783} C_DIS
LIN {X -29.2608,Y 0.5091,Z 60,A 172.5057,B 24.8291,C -3.0152,E1 24.8398,E2 -809.6733} C_DIS
LIN {X -29.2422,Y -1.1522,Z 60,A 176.3276,B 24.8298,C -3.0089,E1 24.8401,E2 -813.5031} C_DIS
LIN {X -29.0979,Y -3.1229,Z 60,A -179.284,B 24.8308,C -3.0005,E1 24.8413,E2 -817.8976} C_DIS
LIN {X -28.5083,Y -6.6112,Z 60,A -173.7233,B 24.8342,C -2.9703,E1 24.8441,E2 -823.4188} C_DIS
LIN {X -28.0853,Y -8.2246,Z 60,A -169.9364,B 24.8349,C -2.9642,E1 24.8469,E2 -827.2131} C_DIS
LIN {X -27.5873,Y -9.7667,Z 60,A -166.8504,B 24.836,C -2.9544,E1 24.8496,E2 -830.2934} C_DIS
LIN {X -26.9428,Y -11.4244,Z 60,A -163.0064,B 24.8368,C -2.9472,E1 24.8537,E2 -834.1414} C_DIS
LIN {X -26.1864,Y -13.0661,Z 60,A -159.6972,B 24.838,C -2.9359,E1 24.8577,E2 -837.4416} C_DIS
LIN {X -25.2359,Y -14.8191,Z 60,A -155.2582,B 24.8387,C -2.9296,E1 24.8638,E2 -841.8887} C_DIS
LIN {X -23.9724,Y -16.7864,Z 60,A -151.1562,B 24.8404,C -2.9148,E1 24.8701,E2 -845.9757} C_DIS
LIN {X -23.0658,Y -18.0109,Z 60,A -148.2141,B 24.8412,C -2.9075,E1 24.8751,E2 -848.9144} C_DIS
LIN {X -22.0401,Y -19.2531,Z 60,A -144.8255,B 24.8417,C -2.9022,E1 24.8812,E2 -852.3059} C_DIS
LIN {X -21.0175,Y -20.3646,Z 60,A -142.2279,B 24.8427,C -2.8932,E1 24.8862,E2 -854.8932} C_DIS
LIN {X -20.026,Y -21.3404,Z 60,A -139.1172,B 24.843,C -2.8907,E1 24.8925,E2 -858.011} C_DIS
LIN {X -18.8602,Y -22.3773,Z 60,A -135.4718,B 24.843,C -2.8898,E1 24.9002,E2 -861.6684} C_DIS
LIN {X -16.5632,Y -24.127,Z 60,A -130.285,B 24.8445,C -2.8766,E1 24.9119,E2 -866.8418} C_DIS
LIN {X -14.752,Y -25.2755,Z 60,A -126.3638,B 24.8454,C -2.8682,E1 24.9212,E2 -870.7551} C_DIS
LIN {X -13.4847,Y -25.9733,Z 60,A -123.5118,B 24.8458,C -2.8648,E1 24.9283,E2 -873.6069} C_DIS
LIN {X -12.1716,Y -26.6137,Z 60,A -120.7947,B 24.8463,C -2.8603,E1 24.9351,E2 -876.3202} C_DIS
LIN {X -11.1366,Y -27.0635,Z 60,A -118.5452,B 24.8465,C -2.8584,E1 24.9409,E2 -878.5704} C_DIS
LIN {X -10.0626,Y -27.4806,Z 60,A -115.951,B 24.8464,C -2.8595,E1 24.9477,E2 -881.1726} C_DIS
LIN {X -7.6805,Y -28.2392,Z 60,A -110.54,B 24.8462,C -2.861,E1 24.9622,E2 -886.5961} C_DIS
LIN {X -5.5006,Y -28.7434,Z 60,A -106.8748,B 24.8471,C -2.8524,E1 24.9722,E2 -890.2451} C_DIS
LIN {X -3.4285,Y -29.0634,Z 60,A -102.0143,B 24.8464,C -2.8589,E1 24.9857,E2 -895.125} C_DIS
LIN {X -1.3125,Y -29.2356,Z 60,A -98.2682,B 24.8469,C -2.855,E1 24.9961,E2 -898.8629} C_DIS
LIN {X 0.0808,Y -29.2633,Z 60,A -96.54,B 24.8479,C -2.8455,E1 25.0009,E2 -900.5685} C_DIS
Enddeposition()
LIN {X 0.0808,Y -29.2633,Z 60,A -96.54,B 24.8479,C -2.8455,E1 25.0009,E2 -900.5685} C_DIS
Startdeposition()
$VEL.CP = VEL_PRINT
LIN {X -0.4652,Y -28.3033,Z 60,A -98.178,B 24.8467,C -2.8567,E1 24.9964,E2 -898.957} C_DIS
LIN {X -2.9998,Y -28.1475,Z 60,A -104.8136,B 24.8481,C -2.843,E1 24.9778,E2 -892.286} C_DIS
LIN {X -5.4194,Y -27.7833,Z 60,A -109.6225,B 24.8478,C -2.846,E1 24.9646,E2 -887.4791} C_DIS
LIN {X -8.94,Y -26.8577,Z 60,A -115.6147,B 24.846,C -2.8626,E1 24.9486,E2 -881.5169} C_DIS
LIN {X -10.7897,Y -26.17,Z 60,A -120.5093,B 24.8465,C -2.8587,E1 24.9358,E2 -876.6026} C_DIS
LIN {X -12.7667,Y -25.2649,Z 60,A -124.6774,B 24.8457,C -2.8657,E1 24.9254,E2 -872.4403} C_DIS
LIN {X -14.5599,Y -24.2754,Z 60,A -128.5648,B 24.8449,C -2.8734,E1 24.916,E2 -868.5597} C_DIS
LIN {X -15.8681,Y -23.4412,Z 60,A -132.4942,B 24.845,C -2.8722,E1 24.9068,E2 -864.6145} C_DIS
LIN {X -18.5167,Y -21.411,Z 60,A -138.4653,B 24.8431,C -2.89,E1 24.8938,E2 -858.6638} C_DIS
LIN {X -19.7735,Y -20.2561,Z 60,A -142.134,B 24.8425,C -2.8953,E1 24.8864,E2 -854.9926} C_DIS
LIN {X -21.1162,Y -18.852,Z 60,A -145.7778,B 24.8413,C -2.9057,E1 24.8795,E2 -851.3578} C_DIS
LIN {X -22.3814,Y -17.3311,Z 60,A -150.824,B 24.8411,C -2.9078,E1 24.8706,E2 -846.2928} C_DIS
LIN {X -24.3267,Y -14.4745,Z 60,A -157.8479,B 24.8392,C -2.9252,E1 24.8601,E2 -839.275} C_DIS
LIN {X -25.5501,Y -12.1851,Z 60,A -162.8036,B 24.8374,C -2.9412,E1 24.8539,E2 -834.3311} C_DIS
LIN {X -26.6183,Y -9.63,Z 60,A -168.689,B 24.8359,C -2.9553,E1 24.8479,E2 -828.4465} C_DIS
LIN {X -27.4455,Y -6.9291,Z 60,A -173.4408,B 24.8333,C -2.9782,E1 24.8443,E2 -823.7218} C_DIS
LIN {X -27.7028,Y -5.8166,Z 60,A -176.5163,B 24.8331,C -2.9804,E1 24.8425,E2 -820.6335} C_DIS
LIN {X -28.1135,Y -3.3022,Z 60,A 178.7262,B 24.831,C -2.9986,E1 24.8406,E2 -815.8912} C_DIS
LIN {X -28.2805,Y -1.2225,Z 60,A 174.0547,B 24.8298,C -3.009,E1 24.8398,E2 -811.2165} C_DIS
LIN {X -28.2931,Y 0.8839,Z 60,A 170.2654,B 24.828,C -3.0251,E1 24.8399,E2 -807.443} C_DIS
LIN {X -28.1858,Y 2.6149,Z 60,A 166.4882,B 24.8269,C -3.0345,E1 24.8407,E2 -803.6656} C_DIS
LIN {X -27.9384,Y 4.5548,Z 60,A 162.4777,B 24.8255,C -3.0465,E1 24.8424,E2 -799.6599} C_DIS
LIN {X -27.534,Y 6.569,Z 60,A 158.3211,B 24.8241,C -3.0593,E1 24.8448,E2 -795.5097} C_DIS
LIN {X -27.0296,Y 8.4072,Z 60,A 154.4562,B 24.8227,C -3.071,E1 24.8479,E2 -791.6505} C_DIS
LIN {X -26.4609,Y 10.0552,Z 60,A 151.0254,B 24.8214,C -3.0822,E1 24.8511,E2 -788.2271} C_DIS
LIN {X -25.627,Y 12.0227,Z 60,A 146.402,B 24.8201,C -3.093,E1 24.8564,E2 -783.6042} C_DIS
LIN {X -24.7911,Y 13.6639,Z 60,A 142.7456,B 24.8188,C -3.1041,E1 24.8612,E2 -779.9548} C_DIS
LIN {X -23.7319,Y 15.4303,Z 60,A 138.701,B 24.8174,C -3.1164,E1 24.8671,E2 -775.9189} C_DIS
LIN {X -22.6986,Y 16.9135,Z 60,A 135.1603,B 24.8162,C -3.1268,E1 24.8729,E2 -772.386} C_DIS
LIN {X -21.608,Y 18.2864,Z 60,A 131.6095,B 24.8151,C -3.1358,E1 24.8791,E2 -768.8403} C_DIS
LIN {X -20.6351,Y 19.3773,Z 60,A 128.9058,B 24.814,C -3.1447,E1 24.8842,E2 -766.1459} C_DIS
LIN {X -19.709,Y 20.3187,Z 60,A 126.0561,B 24.8134,C -3.1498,E1 24.8898,E2 -763.2962} C_DIS
LIN {X -18.8366,Y 21.13,Z 60,A 123.1801,B 24.8132,C -3.152,E1 24.8958,E2 -760.4139} C_DIS
LIN {X -17.4385,Y 22.2978,Z 60,A 119.8313,B 24.812,C -3.1621,E1 24.903,E2 -757.0768} C_DIS
LIN {X -15.9765,Y 23.3673,Z 60,A 115.5751,B 24.8116,C -3.1651,E1 24.9127,E2 -752.813} C_DIS
LIN {X -13.8461,Y 24.6896,Z 60,A 110.8595,B 24.8102,C -3.1767,E1 24.924,E2 -748.1107} C_DIS
LIN {X -12.5104,Y 25.3921,Z 60,A 107.6113,B 24.8098,C -3.18,E1 24.9321,E2 -744.8619} C_DIS
LIN {X -10.7157,Y 26.2004,Z 60,A 103.5187,B 24.8093,C -3.1848,E1 24.9426,E2 -740.7712} C_DIS
LIN {X -8.4053,Y 27.03,Z 60,A 98.7393,B 24.8084,C -3.1921,E1 24.9552,E2 -736.0003} C_DIS
LIN {X -6.3646,Y 27.5821,Z 60,A 94.4031,B 24.8079,C -3.1957,E1 24.967,E2 -731.6665} C_DIS
LIN {X -4.3661,Y 27.9683,Z 60,A 90.0559,B 24.8079,C -3.1968,E1 24.9789,E2 -727.3176} C_DIS
LIN {X -2.4207,Y 28.2031,Z 60,A 86.3351,B 24.8073,C -3.2009,E1 24.9892,E2 -723.6045} C_DIS
LIN {X 0.1725,Y 28.3065,Z 60,A 80.239,B 24.8081,C -3.1948,E1 25.0063,E2 -717.4933} C_DIS
LIN {X 4.1739,Y 27.9979,Z 60,A 71.8746,B 24.8085,C -3.1914,E1 25.0295,E2 -709.1267} C_DIS
LIN {X 6.6197,Y 27.5218,Z 60,A 67.5776,B 24.8079,C -3.196,E1 25.0412,E2 -704.8465} C_DIS
LIN {X 9.0212,Y 26.8307,Z 60,A 62.7944,B 24.808,C -3.195,E1 25.0539,E2 -700.0696} C_DIS
LIN {X 10.8628,Y 26.1396,Z 60,A 58.9833,B 24.8083,C -3.1929,E1 25.0638,E2 -696.2619} C_DIS
LIN {X 12.528,Y 25.3834,Z 60,A 55.223,B 24.8089,C -3.188,E1 25.0733,E2 -692.4998} C_DIS
LIN {X 14.1831,Y 24.4977,Z 60,A 51.4237,B 24.8095,C -3.1829,E1 25.0825,E2 -688.6995} C_DIS
LIN {X 15.7183,Y 23.542,Z 60,A 47.8676,B 24.81,C -3.1784,E1 25.0909,E2 -685.1444} C_DIS
LIN {X 17.3067,Y 22.4002,Z 60,A 43.5384,B 24.8113,C -3.1676,E1 25.1006,E2 -680.8051} C_DIS
LIN {X 18.523,Y 21.4054,Z 60,A 40.7849,B 24.8115,C -3.1664,E1 25.1064,E2 -678.0594} C_DIS
LIN {X 19.9034,Y 20.1281,Z 60,A 36.5827,B 24.8129,C -3.1543,E1 25.1149,E2 -673.8459} C_DIS
LIN {X 21.5492,Y 18.3554,Z 60,A 32.2344,B 24.8134,C -3.1499,E1 25.123,E2 -669.5063} C_DIS
LIN {X 22.5375,Y 17.1282,Z 60,A 28.557,B 24.815,C -3.1367,E1 25.1294,E2 -665.8152} C_DIS
LIN {X 23.6542,Y 15.5488,Z 60,A 24.7822,B 24.8159,C -3.1287,E1 25.1353,E2 -662.04} C_DIS
LIN {X 24.8207,Y 13.6097,Z 60,A 20.674,B 24.8167,C -3.1224,E1 25.141,E2 -657.9381} C_DIS
LIN {X 25.4354,Y 12.4226,Z 60,A 17.894,B 24.8177,C -3.1142,E1 25.1445,E2 -655.1535} C_DIS
LIN {X 26.0641,Y 11.0429,Z 60,A 14.5287,B 24.8191,C -3.1021,E1 25.1483,E2 -651.778} C_DIS
LIN {X 26.8571,Y 8.9419,Z 60,A 10.3265,B 24.8201,C -3.0933,E1 25.1523,E2 -647.5783} C_DIS
LIN {X 27.5572,Y 6.4699,Z 60,A 4.4758,B 24.8228,C -3.0699,E1 25.1564,E2 -641.706} C_DIS
LIN {X 27.9634,Y 4.3983,Z 60,A 0.9896,B 24.8232,C -3.0666,E1 25.1581,E2 -638.2324} C_DIS
LIN {X 28.2198,Y 2.2166,Z 60,A -4.3666,B 24.8261,C -3.0417,E1 25.1596,E2 -632.8488} C_DIS
LIN {X 28.3053,Y -0.1052,Z 60,A -8.2911,B 24.8267,C -3.0367,E1 25.1597,E2 -628.9358} C_DIS
LIN {X 28.2591,Y -1.6413,Z 60,A -11.1706,B 24.8275,C -3.0298,E1 25.1594,E2 -626.0571} C_DIS
LIN {X 28.1517,Y -2.9598,Z 60,A -13.7188,B 24.8282,C -3.023,E1 25.1587,E2 -623.508} C_DIS
LIN {X 28.0072,Y -4.1098,Z 60,A -16.0716,B 24.8291,C -3.0156,E1 25.1579,E2 -621.1514} C_DIS
LIN {X 27.812,Y -5.2701,Z 60,A -18.5004,B 24.83,C -3.0076,E1 25.1567,E2 -618.718} C_DIS
LIN {X 27.5588,Y -6.4653,Z 60,A -20.9261,B 24.8308,C -3.0005,E1 25.1552,E2 -616.2896} C_DIS
LIN {X 27.1527,Y -8.0001,Z 60,A -24.4297,B 24.8323,C -2.9871,E1 25.1526,E2 -612.7743} C_DIS
LIN {X 26.4172,Y -10.1679,Z 60,A -29.6659,B 24.8347,C -2.9658,E1 25.1475,E2 -607.5169} C_DIS
LIN {X 25.5835,Y -12.1155,Z 60,A -33.8868,B 24.836,C -2.954,E1 25.1426,E2 -603.291} C_DIS
LIN {X 24.351,Y -14.4332,Z 60,A -38.4096,B 24.8366,C -2.9485,E1 25.1365,E2 -598.7788} C_DIS
LIN {X 23.5044,Y -15.7744,Z 60,A -41.8155,B 24.8379,C -2.9374,E1 25.1313,E2 -595.3635} C_DIS
LIN {X 22.572,Y -17.0823,Z 60,A -44.7153,B 24.8383,C -2.933,E1 25.1265,E2 -592.4672} C_DIS
LIN {X 21.7937,Y -18.0645,Z 60,A -47.2421,B 24.8391,C -2.9266,E1 25.122,E2 -589.937} C_DIS
LIN {X 20.9766,Y -19.0073,Z 60,A -49.6746,B 24.8396,C -2.9214,E1 25.1175,E2 -587.5031} C_DIS
LIN {X 19.6612,Y -20.3648,Z 60,A -54.2499,B 24.8416,C -2.9036,E1 25.1084,E2 -582.905} C_DIS
LIN {X 18.2501,Y -21.6385,Z 60,A -57.3632,B 24.8416,C -2.9035,E1 25.1019,E2 -579.8038} C_DIS
LIN {X 17.2414,Y -22.4505,Z 60,A -60.0626,B 24.8423,C -2.8971,E1 25.096,E2 -577.0991} C_DIS
LIN {X 16.2251,Y -23.1957,Z 60,A -62.4968,B 24.8427,C -2.8933,E1 25.0905,E2 -574.6644} C_DIS
LIN {X 14.9722,Y -24.0234,Z 60,A -65.8063,B 24.8437,C -2.8845,E1 25.0827,E2 -571.345} C_DIS
LIN {X 13.507,Y -24.8766,Z 60,A -69.4787,B 24.8446,C -2.876,E1 25.0737,E2 -567.663} C_DIS
LIN {X 11.2741,Y -25.9646,Z 60,A -73.753,B 24.8446,C -2.8765,E1 25.0629,E2 -563.4009} C_DIS
LIN {X 9.7095,Y -26.5895,Z 60,A -77.9678,B 24.846,C -2.8633,E1 25.0519,E2 -559.1641} C_DIS
LIN {X 8.0711,Y -27.1318,Z 60,A -81.4189,B 24.8463,C -2.8598,E1 25.0427,E2 -555.7108} C_DIS
LIN {X 5.8118,Y -27.7037,Z 60,A -85.6836,B 24.8463,C -2.86,E1 25.0311,E2 -551.4526} C_DIS
LIN {X 4.28,Y -27.9812,Z 60,A -89.2427,B 24.847,C -2.8536,E1 25.0212,E2 -547.8819} C_DIS
LIN {X 2.1119,Y -28.2277,Z 60,A -93.6835,B 24.8473,C -2.8511,E1 25.0089,E2 -543.4377} C_DIS
LIN {X 0.0724,Y -28.2986,Z 60,A -96.2929,B 24.8458,C -2.8647,E1 25.0017,E2 -540.8613} C_DIS
Enddeposition()
LIN {X 0.0724,Y -28.2986,Z 60,A -96.2929,B 24.8458,C -2.8647,E1 25.0017,E2 -540.8613} C_DIS
Startdeposition()
$VEL.CP = VEL_PRINT
LIN {X 1.2323,Y -27.3205,Z 60,A -93.1593,B 24.8432,C -2.8886,E1 25.0106,E2 -544.0509} C_DIS
LIN {X 3.5469,Y -27.1174,Z 60,A -87.6935,B 24.8423,C -2.8973,E1 25.0258,E2 -549.5336} C_DIS
LIN {X 6.7848,Y -26.4929,Z 60,A -81.1769,B 24.842,C -2.8995,E1 25.0436,E2 -556.0467} C_DIS
LIN {X 9.1039,Y -25.7884,Z 60,A -75.8743,B 24.8411,C -2.9079,E1 25.0576,E2 -561.3591} C_DIS
LIN {X 11.3741,Y -24.8713,Z 60,A -71.4836,B 24.8411,C -2.9073,E1 25.0689,E2 -565.7379} C_DIS
LIN {X 12.7872,Y -24.1753,Z 60,A -68.2631,B 24.8407,C -2.9118,E1 25.0769,E2 -568.9603} C_DIS
LIN {X 14.1019,Y -23.4331,Z 60,A -64.7363,B 24.8396,C -2.9215,E1 25.0854,E2 -572.4992} C_DIS
LIN {X 15.7208,Y -22.379,Z 60,A -60.3839,B 24.8384,C -2.9328,E1 25.0955,E2 -576.8638} C_DIS
LIN {X 17.2076,Y -21.2569,Z 60,A -56.8625,B 24.8379,C -2.9367,E1 25.1032,E2 -580.3812} C_DIS
LIN {X 18.4891,Y -20.1524,Z 60,A -53.692,B 24.8375,C -2.9403,E1 25.1098,E2 -583.5477} C_DIS
LIN {X 19.4534,Y -19.223,Z 60,A -50.6772,B 24.8365,C -2.9494,E1 25.1157,E2 -586.5713} C_DIS
LIN {X 20.6954,Y -17.8793,Z 60,A -46.8253,B 24.8354,C -2.9591,E1 25.1229,E2 -590.429} C_DIS
LIN {X 21.9934,Y -16.2557,Z 60,A -42.6712,B 24.8344,C -2.9681,E1 25.13,E2 -594.5847} C_DIS
LIN {X 23.0529,Y -14.715,Z 60,A -38.4266,B 24.8328,C -2.9827,E1 25.1366,E2 -598.8428} C_DIS
LIN {X 24.1118,Y -12.9071,Z 60,A -34.3431,B 24.8318,C -2.9914,E1 25.1421,E2 -602.9257} C_DIS
LIN {X 24.8517,Y -11.4164,Z 60,A -30.3946,B 24.83,C -3.0072,E1 25.1469,E2 -606.8904} C_DIS
LIN {X 25.821,Y -9.0123,Z 60,A -25.5309,B 24.829,C -3.0165,E1 25.1517,E2 -611.749} C_DIS
LIN {X 26.3526,Y -7.313,Z 60,A -21.3855,B 24.8271,C -3.0331,E1 25.1549,E2 -615.9099} C_DIS
LIN {X 26.7714,Y -5.5903,Z 60,A -18.4092,B 24.8268,C -3.0354,E1 25.1568,E2 -618.8745} C_DIS
Enddeposition()
END
